# B&R Automation Studio project Ampel (part 4)

```cpp
			const TaskStatus h =
				headState.deepPreReact(control, event);
			HFSM2_IF_PLANS(region.headStatus(control) |= h);

			if (!control._consumed)
			HFSM2_IF_PLANS(region.subStatus(control) |=)
			subStates.widePreReact(control, event, active);

			return h;
		} else
	return TaskStatus{};
}

	template <typename TEvent>
	static
	HFSM2_CONSTEXPR(14)
	TaskStatus
	execute(Region& region,
			EventControl& control,
			const TEvent& event) noexcept
	{
		if (!control._consumed) {
HeadState& headState = static_cast<HeadState&>(region);
SubStates& subStates = static_cast<SubStates&>(region);

const TaskStatus h =
	headState.deepPreReact(control, event);
			HFSM2_IF_PLANS(region.headStatus(control) |= h);

			if (!control._consumed)
				HFSM2_IF_PLANS(region.subStatus(control) |=)
					subStates.widePreReact(control, event);

return h;
		} else
			return TaskStatus{};
	}

};

template <typename TRegion>
struct PreReactWrapperT<TRegion, BottomUp> {
	using Region		= TRegion;
	using HeadState		= typename Region::HeadState;
	using SubStates		= typename Region::SubStates;
	using EventControl	= typename Region::EventControl;

	template <typename TEvent>
	static
	HFSM2_CONSTEXPR(14)
	TaskStatus
	execute(Region& region,
	EventControl& control,
	const TEvent& event,
	const Prong active) noexcept
	{
	if (!control._consumed) {
	HeadState& headState = static_cast<HeadState&>(region);
	SubStates& subStates = static_cast<SubStates&>(region);

	const TaskStatus h =
		subStates.widePreReact(control, event, active);
	HFSM2_IF_PLANS(region. subStatus(control) |= h);

	if (!control._consumed)
	HFSM2_IF_PLANS(region.headStatus(control) |=)
	headState.deepPreReact(control, event);

	return h;
} else
			return TaskStatus{};
	}

	template <typename TEvent>
	static
	HFSM2_CONSTEXPR(14)
	TaskStatus
	execute(Region& region,
			EventControl& control,
			const TEvent& event) noexcept
	{
		if (!control._consumed) {
HeadState& headState = static_cast<HeadState&>(region);
SubStates& subStates = static_cast<SubStates&>(region);

const TaskStatus h =
	subStates.widePreReact(control, event);
			HFSM2_IF_PLANS(region. subStatus(control) |= h);

			if (!control._consumed)
				HFSM2_IF_PLANS(region.headStatus(control) |=)
					headState.deepPreReact(control, event);

return h;
		} else
			return TaskStatus{};
	}

};

template <typename, typename>
struct ReactWrapperT;

template <typename TRegion>
struct ReactWrapperT<TRegion, TopDown> {
	using Region		= TRegion;
	using HeadState		= typename Region::HeadState;
	using SubStates		= typename Region::SubStates;
	using EventControl	= typename Region::EventControl;

	template <typename TEvent>
	static
	HFSM2_CONSTEXPR(14)
	TaskStatus
	execute(Region& region,
	EventControl& control,
	const TEvent& event,
	const Prong active) noexcept
	{
	if (!control._consumed) {
	HeadState& headState = static_cast<HeadState&>(region);
	SubStates& subStates = static_cast<SubStates&>(region);

	const TaskStatus h =
		headState.deepReact(control, event);
	HFSM2_IF_PLANS(region.headStatus(control) |= h);

	if (!control._consumed)
	HFSM2_IF_PLANS(region. subStatus(control) |=)
	subStates.wideReact(control, event, active);

	return h;
} else
			return TaskStatus{};
	}

	template <typename TEvent>
	static
	HFSM2_CONSTEXPR(14)
	TaskStatus
	execute(Region& region,
			EventControl& control,
			const TEvent& event) noexcept
	{
		if (!control._consumed) {
HeadState& headState = static_cast<HeadState&>(region);
SubStates& subStates = static_cast<SubStates&>(region);

const TaskStatus h =
	headState.deepReact(control, event);
			HFSM2_IF_PLANS(region.headStatus(control) |= h);

			if (!control._consumed)
				HFSM2_IF_PLANS(region. subStatus(control) |=)
					subStates.wideReact(control, event);

return h;
		} else
			return TaskStatus{};
	}

};

template <typename TRegion>
struct ReactWrapperT<TRegion, BottomUp> {
	using Region		= TRegion;
	using HeadState		= typename Region::HeadState;
	using SubStates		= typename Region::SubStates;
	using EventControl	= typename Region::EventControl;

	template <typename TEvent>
	static
	HFSM2_CONSTEXPR(14)
	TaskStatus
	execute(Region& region,
	EventControl& control,
	const TEvent& event,
	const Prong active) noexcept
	{
	if (!control._consumed) {
	HeadState& headState = static_cast<HeadState&>(region);
	SubStates& subStates = static_cast<SubStates&>(region);

	const TaskStatus h =
		subStates.wideReact(control, event, active);
	HFSM2_IF_PLANS(region. subStatus(control) |= h);

	if (!control._consumed)
	HFSM2_IF_PLANS(region.headStatus(control) |=)
	headState.deepReact(control, event);

	return h;
} else
			return TaskStatus{};
	}

	template <typename TEvent>
	static
	HFSM2_CONSTEXPR(14)
	TaskStatus
	execute(Region& region,
			EventControl& control,
			const TEvent& event) noexcept
	{
		if (!control._consumed) {
HeadState& headState = static_cast<HeadState&>(region);
SubStates& subStates = static_cast<SubStates&>(region);

const TaskStatus h =
	subStates.wideReact(control, event);
			HFSM2_IF_PLANS(region. subStatus(control) |= h);

			if (!control._consumed)
				HFSM2_IF_PLANS(region.headStatus(control) |=)
					headState.deepReact(control, event);

return h;
		} else
			return TaskStatus{};
	}

};

template <typename, typename>
struct PostReactWrapperT;

template <typename TRegion>
struct PostReactWrapperT<TRegion, TopDown> {
	using Region		= TRegion;
	using HeadState		= typename Region::HeadState;
	using SubStates		= typename Region::SubStates;
	using EventControl	= typename Region::EventControl;

	template <typename TEvent>
	static
	HFSM2_CONSTEXPR(14)
	TaskStatus
	execute(Region& region,
	EventControl& control,
	const TEvent& event,
	const Prong active) noexcept
	{
	if (!control._consumed) {
	HeadState& headState = static_cast<HeadState&>(region);
	SubStates& subStates = static_cast<SubStates&>(region);

	HFSM2_IF_PLANS(region. subStatus(control) |=)
	subStates.widePostReact(control, event, active);

	if (control._consumed == false) {
	const TaskStatus h =
		headState.deepPostReact(control, event);
	HFSM2_IF_PLANS(region.headStatus(control) |= h);

	return h;
}
		}

		return TaskStatus{};
	}

	template <typename TEvent>
	static
	HFSM2_CONSTEXPR(14)
	TaskStatus
	execute(Region& region,
			EventControl& control,
			const TEvent& event) noexcept
	{
		if (!control._consumed) {
HeadState& headState = static_cast<HeadState&>(region);
SubStates& subStates = static_cast<SubStates&>(region);

			HFSM2_IF_PLANS(region. subStatus(control) |=)
				subStates.widePostReact(control, event);

			if (control._consumed == false) {
const TaskStatus h =
	headState.deepPostReact(control, event);
				HFSM2_IF_PLANS(region.headStatus(control) |= h);

return h;
			}
		}

		return TaskStatus{};
	}

};

template <typename TRegion>
struct PostReactWrapperT<TRegion, BottomUp> {
	using Region		= TRegion;
	using HeadState		= typename Region::HeadState;
	using SubStates		= typename Region::SubStates;
	using EventControl	= typename Region::EventControl;

	template <typename TEvent>
	static
	HFSM2_CONSTEXPR(14)
	TaskStatus
	execute(Region& region,
	EventControl& control,
	const TEvent& event,
	const Prong active) noexcept
	{
	if (!control._consumed) {
	HeadState& headState = static_cast<HeadState&>(region);
	SubStates& subStates = static_cast<SubStates&>(region);

	HFSM2_IF_PLANS(region.headStatus(control) |=)
	headState.deepPostReact(control, event);

	if (control._consumed == false) {
	const TaskStatus h =
		subStates.widePostReact(control, event, active);
	HFSM2_IF_PLANS(region. subStatus(control) |= h);

	return h;
}
		}

		return TaskStatus{};
	}

	template <typename TEvent>
	static
	HFSM2_CONSTEXPR(14)
	TaskStatus
	execute(Region& region,
			EventControl& control,
			const TEvent& event) noexcept
	{
		if (!control._consumed) {
HeadState& headState = static_cast<HeadState&>(region);
SubStates& subStates = static_cast<SubStates&>(region);

			HFSM2_IF_PLANS(region.headStatus(control) |=)
				headState.deepPostReact(control, event);

			if (control._consumed == false) {
const TaskStatus h =
	subStates.widePostReact(control, event);
				HFSM2_IF_PLANS(region. subStatus(control) |= h);

return h;
			}
		}

		return TaskStatus{};
	}

};

template <typename, typename>
struct QueryWrapperT;

template <typename TRegion>
struct QueryWrapperT<TRegion, TopDown> {
	using Region		= TRegion;
	using HeadState		= typename Region::HeadState;
	using SubStates		= typename Region::SubStates;
	using ConstControl	= typename Region::ConstControl;

	template <typename TEvent>
	static
	HFSM2_CONSTEXPR(14)
	void
	execute(const Region& region,
	ConstControl& control,
	TEvent& event,
	const Prong active) noexcept
	{
	const HeadState& headState = static_cast<const HeadState&>(region);
	const SubStates& subStates = static_cast<const SubStates&>(region);

	if (!control._consumed)
	headState.deepQuery(control, event);

	if (!control._consumed)
	subStates.wideQuery(control, event, active);
}

	template <typename TEvent>
	static
	HFSM2_CONSTEXPR(14)
	void
	execute(const Region& region,
			ConstControl& control,
			TEvent& event) noexcept
	{
const HeadState& headState = static_cast<const HeadState&>(region);
const SubStates& subStates = static_cast<const SubStates&>(region);

		if (!control._consumed)
			headState.deepQuery(control, event);

		if (!control._consumed)
			subStates.wideQuery(control, event);
	}

};

template <typename TRegion>
struct QueryWrapperT<TRegion, BottomUp> {
	using Region		= TRegion;
	using HeadState		= typename Region::HeadState;
	using SubStates		= typename Region::SubStates;
	using ConstControl	= typename Region::ConstControl;

	template <typename TEvent>
	static
	HFSM2_CONSTEXPR(14)
	void
	execute(const Region& region,
	ConstControl& control,
	TEvent& event,
	const Prong active) noexcept
	{
	const HeadState& headState = static_cast<const HeadState&>(region);
	const SubStates& subStates = static_cast<const SubStates&>(region);

	if (!control._consumed)
	subStates.wideQuery(control, event, active);

	if (!control._consumed)
	headState.deepQuery(control, event);
}

	template <typename TEvent>
	static
	HFSM2_CONSTEXPR(14)
	void
	execute(const Region& region,
			ConstControl& control,
			TEvent& event) noexcept
	{
const HeadState& headState = static_cast<const HeadState&>(region);
const SubStates& subStates = static_cast<const SubStates&>(region);

		if (!control._consumed)
			subStates.wideQuery(control, event);

		if (!control._consumed)
			headState.deepQuery(control, event);
	}

};

}
}

namespace hfsm2 {
	namespace detail {

		template <
		typename TIndices
		, typename TArgs
		, Strategy TStrategy
		, Prong NProng
		, typename... TStates
		>
		struct HFSM2_EMPTY_BASES CS_<
			TIndices
			, TArgs
			, TStrategy
			, NProng
			, TL_<TStates...>
		>
		:					 LHalfCS<
		TIndices
		, TArgs
		, TStrategy
		, NProng
		, TL_<TStates...>
		>
		,					 RHalfCS<
		TIndices
		, TArgs
		, TStrategy
		, NProng
		, TL_<TStates...>
		>
		{
		static_assert(sizeof...(TStates) >= 2, "");

		using Indices		= TIndices;
		static constexpr StateID  INITIAL_ID  = Indices::STATE_ID;
		static constexpr Short	  COMPO_INDEX = Indices::COMPO_INDEX;
		static constexpr Short	  ORTHO_INDEX = Indices::ORTHO_INDEX;
		static constexpr Short	  ORTHO_UNIT  = Indices::ORTHO_UNIT;

		static constexpr Strategy STRATEGY	  = TStrategy;

		static constexpr RegionID REGION_ID	  = COMPO_INDEX + ORTHO_INDEX;
		static constexpr Prong	  PRONG_INDEX = NProng;

		using Args			= TArgs;
		using SubStateList	= TL_<TStates...>;

#if HFSM2_UTILITY_THEORY_AVAILABLE()
		using Rank			= typename Args::Rank;
		using Utility		= typename Args::Utility;
		using UP			= typename Args::UP;
#endif

		using StateList		= typename Args::StateList;
		using RegionList	= typename Args::RegionList;

		using Registry		= RegistryT<Args>;
		using StateParents	= typename Registry::StateParents;

		using ConstControl	= ConstControlT<Args>;
		using Control		= ControlT	   <Args>;
		using PlanControl	= PlanControlT <Args>;
		using FullControl	= FullControlT <Args>;
		using GuardControl	= GuardControlT<Args>;
		using EventControl	= EventControlT<Args>;

		using LStateList	= LHalfTypes<TStates...>;
		using LHalfInfo		= CSI_<LStateList>;

		static constexpr Prong	  L_PRONG	  = PRONG_INDEX;
		static constexpr Prong	  R_PRONG	  = PRONG_INDEX + LStateList::SIZE;

		using LHalf			= LHalfCS<
			Indices
			, Args
			, STRATEGY
			, PRONG_INDEX
			, SubStateList
			>;

		using RHalf			= RHalfCS<
			Indices
			, Args
			, STRATEGY
			, PRONG_INDEX
			, SubStateList
			>;

		HFSM2_CONSTEXPR(14)	void		wideRegister			   (Registry& registry, const Parent parent)								noexcept;

		HFSM2_CONSTEXPR(14)	bool		wideForwardEntryGuard	   (GuardControl& control,						  const Prong prong)		noexcept;
		HFSM2_CONSTEXPR(14)	bool		wideEntryGuard			   (GuardControl& control,						  const Prong prong)		noexcept;

		HFSM2_CONSTEXPR(14)	void		wideEnter				   ( PlanControl& control,						  const Prong prong)		noexcept;
		HFSM2_CONSTEXPR(14)	void		wideReenter				   ( PlanControl& control,						  const Prong prong)		noexcept;

		HFSM2_CONSTEXPR(14)	TaskStatus	widePreUpdate			   ( FullControl& control,						  const Prong prong)		noexcept;
		HFSM2_CONSTEXPR(14)	TaskStatus	wideUpdate				   ( FullControl& control,						  const Prong prong)		noexcept;
		HFSM2_CONSTEXPR(14)	TaskStatus	widePostUpdate			   ( FullControl& control,						  const Prong prong)		noexcept;

		template <typename TEvent>
		HFSM2_CONSTEXPR(14)	TaskStatus	widePreReact			   (EventControl& control, const TEvent& event,	  const Prong prong)		noexcept;

		template <typename TEvent>
		HFSM2_CONSTEXPR(14)	TaskStatus	wideReact				   (EventControl& control, const TEvent& event,	  const Prong prong)		noexcept;

		template <typename TEvent>
		HFSM2_CONSTEXPR(14)	TaskStatus	widePostReact			   (EventControl& control, const TEvent& event,	  const Prong prong)		noexcept;

		template <typename TEvent>
		HFSM2_CONSTEXPR(14)	void		wideQuery				   (ConstControl& control,		 TEvent& event,	  const Prong prong)  const noexcept;

#if HFSM2_PLANS_AVAILABLE()
		HFSM2_CONSTEXPR(14)	TaskStatus	wideUpdatePlans			   ( FullControl& control,						  const Prong prong)		noexcept;
#endif

		HFSM2_CONSTEXPR(14)	bool		wideForwardExitGuard	   (GuardControl& control,						  const Prong prong)		noexcept;
		HFSM2_CONSTEXPR(14)	bool		wideExitGuard			   (GuardControl& control,						  const Prong prong)		noexcept;

		HFSM2_CONSTEXPR(14)	void		wideExit				   ( PlanControl& control,						  const Prong prong)		noexcept;

		HFSM2_CONSTEXPR(14)	void		wideForwardActive		   (	 Control& control, const Request request, const Prong prong)		noexcept;
		HFSM2_CONSTEXPR(14)	void		wideForwardRequest		   (	 Control& control, const Request request, const Prong prong)		noexcept;

		HFSM2_CONSTEXPR(14)	void		wideRequestChangeComposite (	 Control& control, const Request request				   )		noexcept;
		HFSM2_CONSTEXPR(14)	void		wideRequestChangeResumable (	 Control& control, const Request request, const Prong prong)		noexcept;
		HFSM2_CONSTEXPR(14)	void		wideRequestChangeSelectable(	 Control& control, const Request request, const Prong prong)		noexcept;

		HFSM2_CONSTEXPR(14)	void		wideRequestRestart		   (	 Control& control, const Request request				   )		noexcept;
		HFSM2_CONSTEXPR(14)	void		wideRequestResume		   (	 Control& control, const Request request, const Prong prong)		noexcept;
		HFSM2_CONSTEXPR(14)	void		wideRequestSelect		   (	 Control& control, const Request request, const Prong prong)		noexcept;

#if HFSM2_UTILITY_THEORY_AVAILABLE()
		HFSM2_CONSTEXPR(14)	UP			wideReportChangeComposite  (	 Control& control																  )		noexcept;
		HFSM2_CONSTEXPR(14)	UP			wideReportChangeResumable  (	 Control& control,						  const Prong prong						  )		noexcept;
		HFSM2_CONSTEXPR(14)	UP			wideReportChangeSelectable (	 Control& control,						  const Prong prong						  )		noexcept;
		HFSM2_CONSTEXPR(14)	UP			wideReportChangeUtilitarian(	 Control& control																  )		noexcept;
		HFSM2_CONSTEXPR(14)	Utility		wideReportChangeRandom	   (	 Control& control, Utility* const options, const Rank* const ranks, const Rank top)		noexcept;

		HFSM2_CONSTEXPR(14)	UP			wideReportUtilize		   (	 Control& control																  )		noexcept;
		HFSM2_CONSTEXPR(14)	Rank		wideReportRank			   (	 Control& control,								 Rank* const ranks				  )		noexcept;
		HFSM2_CONSTEXPR(14)	Utility		wideReportRandomize		   (	 Control& control, Utility* const options, const Rank* const ranks, const Rank top)		noexcept;
#endif

		HFSM2_CONSTEXPR(14)	void		wideChangeToRequested	   ( PlanControl& control,						  const Prong prong)		noexcept;

#if HFSM2_SERIALIZATION_AVAILABLE()
		using WriteStream	= typename Args::WriteStream;
		using ReadStream	= typename Args::ReadStream;

		HFSM2_CONSTEXPR(14)	void		wideSaveActive			   (const Registry& registry, WriteStream& stream, const Prong prong)  const noexcept;
		HFSM2_CONSTEXPR(14)	void		wideSaveResumable		   (const Registry& registry, WriteStream& stream					)  const noexcept;

		HFSM2_CONSTEXPR(14)	void		wideLoadRequested		   (      Registry& registry,  ReadStream& stream, const Prong prong)  const noexcept;
		HFSM2_CONSTEXPR(14)	void		wideLoadResumable		   (      Registry& registry,  ReadStream& stream					)  const noexcept;
#endif

#if HFSM2_STRUCTURE_REPORT_AVAILABLE()
		using StructureStateInfos = typename Args::StructureStateInfos;

		static constexpr Long NAME_COUNT = LHalf::NAME_COUNT + RHalf::NAME_COUNT;

		HFSM2_CONSTEXPR(14)	void wideGetNames(const Long parent,
		const RegionType region,
		const Short depth,
		StructureStateInfos& stateInfos)	  const noexcept;
#endif

	};

}
}

namespace hfsm2 {
	namespace detail {

		template <typename TN_, typename TA_, Strategy SG_, Prong NP_, typename... TS_>
		HFSM2_CONSTEXPR(14)
		void
			CS_<TN_, TA_, SG_, NP_, TL_<TS_...>>::wideRegister(Registry& registry,
		const Parent parent) noexcept
		{
		LHalf::wideRegister(registry, Parent{parent.forkId, L_PRONG});
		RHalf::wideRegister(registry, Parent{parent.forkId, R_PRONG});
	}

	template <typename TN_, typename TA_, Strategy SG_, Prong NP_, typename... TS_>
	HFSM2_CONSTEXPR(14)
	bool
		CS_<TN_, TA_, SG_, NP_, TL_<TS_...>>::wideForwardEntryGuard(GuardControl& control,
	const Prong prong) noexcept
	{
	HFSM2_ASSERT(prong != INVALID_SHORT);

	if (prong < R_PRONG)
	return LHalf::wideForwardEntryGuard(control, prong);
	else
	return RHalf::wideForwardEntryGuard(control, prong);
}

template <typename TN_, typename TA_, Strategy SG_, Prong NP_, typename... TS_>
HFSM2_CONSTEXPR(14)
bool
	CS_<TN_, TA_, SG_, NP_, TL_<TS_...>>::wideEntryGuard(GuardControl& control,
													 const Prong prong) noexcept
{
	HFSM2_ASSERT(prong != INVALID_PRONG);

	if (prong < R_PRONG)
		return LHalf::wideEntryGuard(control, prong);
	else
		return RHalf::wideEntryGuard(control, prong);
}

template <typename TN_, typename TA_, Strategy SG_, Prong NP_, typename... TS_>
HFSM2_CONSTEXPR(14)
void
	CS_<TN_, TA_, SG_, NP_, TL_<TS_...>>::wideEnter(PlanControl& control,
												const Prong prong) noexcept
{
	HFSM2_ASSERT(prong != INVALID_PRONG);

	if (prong < R_PRONG)
		LHalf::wideEnter(control, prong);
	else
		RHalf::wideEnter(control, prong);
}

template <typename TN_, typename TA_, Strategy SG_, Prong NP_, typename... TS_>
HFSM2_CONSTEXPR(14)
void
	CS_<TN_, TA_, SG_, NP_, TL_<TS_...>>::wideReenter(PlanControl& control,
												  const Prong prong) noexcept
{
	HFSM2_ASSERT(prong != INVALID_PRONG);

	if (prong < R_PRONG)
		LHalf::wideReenter(control, prong);
	else
		RHalf::wideReenter(control, prong);
}

template <typename TN_, typename TA_, Strategy SG_, Prong NP_, typename... TS_>
HFSM2_CONSTEXPR(14)
TaskStatus
	CS_<TN_, TA_, SG_, NP_, TL_<TS_...>>::widePreUpdate(FullControl& control,
													const Prong prong) noexcept
{
	HFSM2_ASSERT(prong != INVALID_PRONG);

	return prong < R_PRONG ?
		LHalf::widePreUpdate(control, prong) :
		RHalf::widePreUpdate(control, prong);
}

template <typename TN_, typename TA_, Strategy SG_, Prong NP_, typename... TS_>
HFSM2_CONSTEXPR(14)
TaskStatus
	CS_<TN_, TA_, SG_, NP_, TL_<TS_...>>::wideUpdate(FullControl& control,
												 const Prong prong) noexcept
{
	HFSM2_ASSERT(prong != INVALID_PRONG);

	return prong < R_PRONG ?
		LHalf::wideUpdate(control, prong) :
		RHalf::wideUpdate(control, prong);
}

template <typename TN_, typename TA_, Strategy SG_, Prong NP_, typename... TS_>
HFSM2_CONSTEXPR(14)
TaskStatus
	CS_<TN_, TA_, SG_, NP_, TL_<TS_...>>::widePostUpdate(FullControl& control,
													 const Prong prong) noexcept
{
	HFSM2_ASSERT(prong != INVALID_PRONG);

	return prong < R_PRONG ?
		LHalf::widePostUpdate(control, prong) :
		RHalf::widePostUpdate(control, prong);
}

template <typename TN_, typename TA_, Strategy SG_, Prong NP_, typename... TS_>
template <typename TEvent>
HFSM2_CONSTEXPR(14)
TaskStatus
	CS_<TN_, TA_, SG_, NP_, TL_<TS_...>>::widePreReact(EventControl& control,
												   const TEvent& event,
												   const Prong prong) noexcept
{
	HFSM2_ASSERT(prong != INVALID_PRONG);

	return prong < R_PRONG ?
		LHalf::widePreReact(control, event, prong) :
		RHalf::widePreReact(control, event, prong);
}

template <typename TN_, typename TA_, Strategy SG_, Prong NP_, typename... TS_>
template <typename TEvent>
HFSM2_CONSTEXPR(14)
TaskStatus
	CS_<TN_, TA_, SG_, NP_, TL_<TS_...>>::wideReact(EventControl& control,
												const TEvent& event,
												const Prong prong) noexcept
{
	HFSM2_ASSERT(prong != INVALID_PRONG);

	return prong < R_PRONG ?
		LHalf::wideReact(control, event, prong) :
		RHalf::wideReact(control, event, prong);
}

template <typename TN_, typename TA_, Strategy SG_, Prong NP_, typename... TS_>
template <typename TEvent>
HFSM2_CONSTEXPR(14)
TaskStatus
	CS_<TN_, TA_, SG_, NP_, TL_<TS_...>>::widePostReact(EventControl& control,
													const TEvent& event,
													const Prong prong) noexcept
{
	HFSM2_ASSERT(prong != INVALID_PRONG);

	return prong < R_PRONG ?
		LHalf::widePostReact(control, event, prong) :
		RHalf::widePostReact(control, event, prong);
}

template <typename TN_, typename TA_, Strategy SG_, Prong NP_, typename... TS_>
template <typename TEvent>
HFSM2_CONSTEXPR(14)
void
	CS_<TN_, TA_, SG_, NP_, TL_<TS_...>>::wideQuery(ConstControl& control,
												TEvent& event,
												const Prong prong) const noexcept
{
	HFSM2_ASSERT(prong != INVALID_PRONG);

	return prong < R_PRONG ?
		LHalf::wideQuery(control, event, prong) :
		RHalf::wideQuery(control, event, prong);
}

#if HFSM2_PLANS_AVAILABLE()

template <typename TN_, typename TA_, Strategy SG_, Prong NP_, typename... TS_>
HFSM2_CONSTEXPR(14)
TaskStatus
	CS_<TN_, TA_, SG_, NP_, TL_<TS_...>>::wideUpdatePlans(FullControl& control,
													  const Prong prong) noexcept
{
	HFSM2_ASSERT(prong != INVALID_PRONG);

	return prong < R_PRONG ?
		LHalf::wideUpdatePlans(control, prong) :
		RHalf::wideUpdatePlans(control, prong);
}

#endif

template <typename TN_, typename TA_, Strategy SG_, Prong NP_, typename... TS_>
HFSM2_CONSTEXPR(14)
bool
	CS_<TN_, TA_, SG_, NP_, TL_<TS_...>>::wideForwardExitGuard(GuardControl& control,
														   const Prong prong) noexcept
{
	HFSM2_ASSERT(prong != INVALID_PRONG);

	if (prong < R_PRONG)
		return LHalf::wideForwardExitGuard(control, prong);
	else
		return RHalf::wideForwardExitGuard(control, prong);
}

template <typename TN_, typename TA_, Strategy SG_, Prong NP_, typename... TS_>
HFSM2_CONSTEXPR(14)
bool
	CS_<TN_, TA_, SG_, NP_, TL_<TS_...>>::wideExitGuard(GuardControl& control,
													const Prong prong) noexcept
{
	HFSM2_ASSERT(prong != INVALID_PRONG);

	if (prong < R_PRONG)
		return LHalf::wideExitGuard(control, prong);
	else
		return RHalf::wideExitGuard(control, prong);
}

template <typename TN_, typename TA_, Strategy SG_, Prong NP_, typename... TS_>
HFSM2_CONSTEXPR(14)
void
	CS_<TN_, TA_, SG_, NP_, TL_<TS_...>>::wideExit(PlanControl& control,
											   const Prong prong) noexcept
{
	HFSM2_ASSERT(prong != INVALID_PRONG);

	if (prong < R_PRONG)
		LHalf::wideExit(control, prong);
	else
		RHalf::wideExit(control, prong);
}

template <typename TN_, typename TA_, Strategy SG_, Prong NP_, typename... TS_>
HFSM2_CONSTEXPR(14)
void
	CS_<TN_, TA_, SG_, NP_, TL_<TS_...>>::wideForwardActive(Control& control,
														const Request request,
														const Prong prong) noexcept
{
	HFSM2_ASSERT(prong != INVALID_PRONG);

	if (prong < R_PRONG)
		LHalf::wideForwardActive(control, request, prong);
	else
		RHalf::wideForwardActive(control, request, prong);
}

template <typename TN_, typename TA_, Strategy SG_, Prong NP_, typename... TS_>
HFSM2_CONSTEXPR(14)
void
	CS_<TN_, TA_, SG_, NP_, TL_<TS_...>>::wideForwardRequest(Control& control,
														 const Request request,
														 const Prong prong) noexcept
{
	HFSM2_ASSERT(prong != INVALID_PRONG);

	if (prong < R_PRONG)
		LHalf::wideForwardRequest(control, request, prong);
	else
		RHalf::wideForwardRequest(control, request, prong);
}

template <typename TN_, typename TA_, Strategy SG_, Prong NP_, typename... TS_>
HFSM2_CONSTEXPR(14)
void
	CS_<TN_, TA_, SG_, NP_, TL_<TS_...>>::wideRequestChangeComposite(Control& control,
																 const Request request) noexcept
{
	LHalf::wideRequestChangeComposite(control, request);
}

template <typename TN_, typename TA_, Strategy SG_, Prong NP_, typename... TS_>
HFSM2_CONSTEXPR(14)
void
	CS_<TN_, TA_, SG_, NP_, TL_<TS_...>>::wideRequestChangeResumable(Control& control,
																 const Request request,
																 const Prong prong) noexcept
{
	HFSM2_ASSERT(prong != INVALID_PRONG);

	if (prong < R_PRONG)
		LHalf::wideRequestChangeResumable(control, request, prong);
	else
		RHalf::wideRequestChangeResumable(control, request, prong);
}

template <typename TN_, typename TA_, Strategy SG_, Prong NP_, typename... TS_>
HFSM2_CONSTEXPR(14)
void
	CS_<TN_, TA_, SG_, NP_, TL_<TS_...>>::wideRequestChangeSelectable(Control& control,
																  const Request request,
																  const Prong prong) noexcept
{
	HFSM2_ASSERT(prong != INVALID_PRONG);

	if (prong < R_PRONG)
		LHalf::wideRequestChangeSelectable(control, request, prong);
	else
		RHalf::wideRequestChangeSelectable(control, request, prong);
}

template <typename TN_, typename TA_, Strategy SG_, Prong NP_, typename... TS_>
HFSM2_CONSTEXPR(14)
void
	CS_<TN_, TA_, SG_, NP_, TL_<TS_...>>::wideRequestRestart(Control& control,
														 const Request request) noexcept
{
	LHalf::wideRequestRestart(control, request);
}

template <typename TN_, typename TA_, Strategy SG_, Prong NP_, typename... TS_>
HFSM2_CONSTEXPR(14)
void
	CS_<TN_, TA_, SG_, NP_, TL_<TS_...>>::wideRequestResume(Control& control,
														const Request request,
														const Prong prong) noexcept
{
	HFSM2_ASSERT(prong != INVALID_PRONG);

	if (prong < R_PRONG)
		LHalf::wideRequestResume(control, request, prong);
	else
		RHalf::wideRequestResume(control, request, prong);
}

template <typename TN_, typename TA_, Strategy SG_, Prong NP_, typename... TS_>
HFSM2_CONSTEXPR(14)
void
	CS_<TN_, TA_, SG_, NP_, TL_<TS_...>>::wideRequestSelect(Control& control,
														const Request request,
														const Prong prong) noexcept
{
	HFSM2_ASSERT(prong != INVALID_PRONG);

	if (prong < R_PRONG)
		LHalf::wideRequestSelect(control, request, prong);
	else
		RHalf::wideRequestSelect(control, request, prong);
}

#if HFSM2_UTILITY_THEORY_AVAILABLE()

template <typename TN_, typename TA_, Strategy SG_, Prong NP_, typename... TS_>
HFSM2_CONSTEXPR(14)
typename TA_::UP
	CS_<TN_, TA_, SG_, NP_, TL_<TS_...>>::wideReportUtilize(Control& control) noexcept {
const UP l = LHalf::wideReportUtilize(control);
const UP r = RHalf::wideReportUtilize(control);

	return l.utility >= r.utility ?
l : r;
}

template <typename TN_, typename TA_, Strategy SG_, Prong NP_, typename... TS_>
HFSM2_CONSTEXPR(14)
typename TA_::Rank
	CS_<TN_, TA_, SG_, NP_, TL_<TS_...>>::wideReportRank(Control& control,
													 Rank* const ranks) noexcept
{
	HFSM2_ASSERT(ranks);

const Rank l = LHalf::wideReportRank(control, ranks);
const Rank r = RHalf::wideReportRank(control, ranks + LStateList::SIZE);

	return l >= r ?
l : r;
}

template <typename TN_, typename TA_, Strategy SG_, Prong NP_, typename... TS_>
HFSM2_CONSTEXPR(14)
typename TA_::Utility
	CS_<TN_, TA_, SG_, NP_, TL_<TS_...>>::wideReportRandomize(Control& control,
														  Utility* const utilities,
														  const Rank* const ranks,
														  const Rank top) noexcept
{
	HFSM2_ASSERT(utilities && ranks);

const Utility l = LHalf::wideReportRandomize(control, utilities,					ranks,					  top);
const Utility r = RHalf::wideReportRandomize(control, utilities + LStateList::SIZE, ranks + LStateList::SIZE, top);

	return { l + r };
}

template <typename TN_, typename TA_, Strategy SG_, Prong NP_, typename... TS_>
HFSM2_CONSTEXPR(14)
typename TA_::UP
	CS_<TN_, TA_, SG_, NP_, TL_<TS_...>>::wideReportChangeComposite(Control& control) noexcept {
	return LHalf::wideReportChangeComposite(control);
}

template <typename TN_, typename TA_, Strategy SG_, Prong NP_, typename... TS_>
HFSM2_CONSTEXPR(14)
typename TA_::UP
	CS_<TN_, TA_, SG_, NP_, TL_<TS_...>>::wideReportChangeResumable(Control& control,
																const Prong prong) noexcept
{
	HFSM2_ASSERT(prong != INVALID_PRONG);

	if (prong < R_PRONG)
		return LHalf::wideReportChangeResumable(control, prong);
	else
		return RHalf::wideReportChangeResumable(control, prong);
}

template <typename TN_, typename TA_, Strategy SG_, Prong NP_, typename... TS_>
HFSM2_CONSTEXPR(14)
typename TA_::UP
	CS_<TN_, TA_, SG_, NP_, TL_<TS_...>>::wideReportChangeSelectable(Control& control,
																 const Prong prong) noexcept
{
	HFSM2_ASSERT(prong != INVALID_PRONG);

	if (prong < R_PRONG)
		return LHalf::wideReportChangeSelectable(control, prong);
	else
		return RHalf::wideReportChangeSelectable(control, prong);
}

template <typename TN_, typename TA_, Strategy SG_, Prong NP_, typename... TS_>
HFSM2_CONSTEXPR(14)
typename TA_::UP
	CS_<TN_, TA_, SG_, NP_, TL_<TS_...>>::wideReportChangeUtilitarian(Control& control) noexcept {
const UP l = LHalf::wideReportChangeUtilitarian(control);
const UP r = RHalf::wideReportChangeUtilitarian(control);

	return l.utility >= r.utility ?
l : r;
}

template <typename TN_, typename TA_, Strategy SG_, Prong NP_, typename... TS_>
HFSM2_CONSTEXPR(14)
typename TA_::Utility
	CS_<TN_, TA_, SG_, NP_, TL_<TS_...>>::wideReportChangeRandom(Control& control,
															 Utility* const utilities,
															 const Rank* const ranks,
															 const Rank top) noexcept
{
	HFSM2_ASSERT(utilities && ranks);

const Utility l = LHalf::wideReportChangeRandom(control, utilities,					   ranks,					 top);
const Utility r = RHalf::wideReportChangeRandom(control, utilities + LStateList::SIZE, ranks + LStateList::SIZE, top);

	return { l + r };
}

#endif

template <typename TN_, typename TA_, Strategy SG_, Prong NP_, typename... TS_>
HFSM2_CONSTEXPR(14)
void
	CS_<TN_, TA_, SG_, NP_, TL_<TS_...>>::wideChangeToRequested(PlanControl& control,
															const Prong prong) noexcept
{
	HFSM2_ASSERT(prong != INVALID_PRONG);

	if (prong < R_PRONG)
		LHalf::wideChangeToRequested(control, prong);
	else
		RHalf::wideChangeToRequested(control, prong);
}

#if HFSM2_SERIALIZATION_AVAILABLE()

template <typename TN_, typename TA_, Strategy SG_, Prong NP_, typename... TS_>
HFSM2_CONSTEXPR(14)
void
	CS_<TN_, TA_, SG_, NP_, TL_<TS_...>>::wideSaveActive(const Registry& registry,
													 WriteStream& stream,
													 const Prong prong) const noexcept
{
	HFSM2_ASSERT(prong != INVALID_PRONG);

	if (prong < R_PRONG) {
		LHalf::wideSaveActive   (registry, stream, prong);
		RHalf::wideSaveResumable(registry, stream);
	} else {
		LHalf::wideSaveResumable(registry, stream);
		RHalf::wideSaveActive   (registry, stream, prong);
	}
}

template <typename TN_, typename TA_, Strategy SG_, Prong NP_, typename... TS_>
HFSM2_CONSTEXPR(14)
void
	CS_<TN_, TA_, SG_, NP_, TL_<TS_...>>::wideSaveResumable(const Registry& registry,
														WriteStream& stream) const noexcept
{
	LHalf::wideSaveResumable(registry, stream);
	RHalf::wideSaveResumable(registry, stream);
}

template <typename TN_, typename TA_, Strategy SG_, Prong NP_, typename... TS_>
HFSM2_CONSTEXPR(14)
void
	CS_<TN_, TA_, SG_, NP_, TL_<TS_...>>::wideLoadRequested(Registry& registry,
														ReadStream& stream,
														const Prong prong) const noexcept
{
	HFSM2_ASSERT(prong != INVALID_PRONG);

	if (prong < R_PRONG) {
		LHalf::wideLoadRequested(registry, stream, prong);
		RHalf::wideLoadResumable(registry, stream);
	} else {
		LHalf::wideLoadResumable(registry, stream);
		RHalf::wideLoadRequested(registry, stream, prong);
	}
}

template <typename TN_, typename TA_, Strategy SG_, Prong NP_, typename... TS_>
HFSM2_CONSTEXPR(14)
void
	CS_<TN_, TA_, SG_, NP_, TL_<TS_...>>::wideLoadResumable(Registry& registry,
														ReadStream& stream) const noexcept
{
	LHalf::wideLoadResumable(registry, stream);
	RHalf::wideLoadResumable(registry, stream);
}

#endif

#if HFSM2_STRUCTURE_REPORT_AVAILABLE()

template <typename TN_, typename TA_, Strategy SG_, Prong NP_, typename... TS_>
HFSM2_CONSTEXPR(14)
void
	CS_<TN_, TA_, SG_, NP_, TL_<TS_...>>::wideGetNames(const Long parent,
												   const RegionType /*region*/,
												   const Short depth,
												   StructureStateInfos& stateInfos) const noexcept
{
	LHalf::wideGetNames(parent, RegionType::COMPOSITE, depth, stateInfos);
	RHalf::wideGetNames(parent, RegionType::COMPOSITE, depth, stateInfos);
}

#endif

}
}

namespace hfsm2 {
	namespace detail {

		template <
		typename TIndices
		, typename TArgs
		, Strategy TStrategy
		, Prong NProng
		, typename TState
		>
		struct HFSM2_EMPTY_BASES CS_<
			TIndices
			, TArgs
			, TStrategy
			, NProng
			, TL_<TState>
			>
			:					 MaterialT<
			TIndices
			, TArgs
			, TState
			>
			{
			using Indices		= TIndices;
			static constexpr StateID  INITIAL_ID  = Indices::STATE_ID;
			static constexpr Short	  COMPO_INDEX = Indices::COMPO_INDEX;
			static constexpr Short	  ORTHO_INDEX = Indices::ORTHO_INDEX;
			static constexpr Short	  ORTHO_UNIT  = Indices::ORTHO_UNIT;

			static constexpr Strategy STRATEGY	  = TStrategy;

			static constexpr RegionID REGION_ID	  = COMPO_INDEX + ORTHO_INDEX;
			static constexpr Prong	  PRONG_INDEX = NProng;

			using Args			= TArgs;

#if HFSM2_UTILITY_THEORY_AVAILABLE()
			using Rank			= typename Args::Rank;
			using Utility		= typename Args::Utility;
			using UP			= typename Args::UP;
#endif

			using StateList		= typename Args::StateList;
			using RegionList	= typename Args::RegionList;

			using Registry		= RegistryT<Args>;
			using StateParents	= typename Registry::StateParents;

			using ConstControl	= ConstControlT<Args>;
			using Control		= ControlT	   <Args>;
			using PlanControl	= PlanControlT <Args>;
			using FullControl	= FullControlT <Args>;
			using GuardControl	= GuardControlT<Args>;
			using EventControl	= EventControlT<Args>;

			using Single		= MaterialT<
				Indices
				, Args
				, TState
				>;

			HFSM2_CONSTEXPR(14)	void		wideRegister			   (Registry& registry, const Parent parent)								noexcept;

			HFSM2_CONSTEXPR(14)	bool		wideForwardEntryGuard	   (GuardControl& control,						  const Prong prong)		noexcept;
			HFSM2_CONSTEXPR(14)	bool		wideEntryGuard			   (GuardControl& control,						  const Prong prong)		noexcept;

			HFSM2_CONSTEXPR(14)	void		wideEnter				   ( PlanControl& control,						  const Prong prong)		noexcept;
			HFSM2_CONSTEXPR(14)	void		wideReenter				   ( PlanControl& control,						  const Prong prong)		noexcept;

			HFSM2_CONSTEXPR(14)	TaskStatus	widePreUpdate			   ( FullControl& control,						  const Prong prong)		noexcept;
			HFSM2_CONSTEXPR(14)	TaskStatus	wideUpdate				   ( FullControl& control,						  const Prong prong)		noexcept;
			HFSM2_CONSTEXPR(14)	TaskStatus	widePostUpdate			   ( FullControl& control,						  const Prong prong)		noexcept;

			template <typename TEvent>
			HFSM2_CONSTEXPR(14)	TaskStatus	widePreReact			   (EventControl& control, const TEvent& event,	  const Prong prong)		noexcept;

			template <typename TEvent>
			HFSM2_CONSTEXPR(14)	TaskStatus	wideReact				   (EventControl& control, const TEvent& event,	  const Prong prong)		noexcept;

			template <typename TEvent>
			HFSM2_CONSTEXPR(14)	TaskStatus	widePostReact			   (EventControl& control, const TEvent& event,	  const Prong prong)		noexcept;

			template <typename TEvent>
			HFSM2_CONSTEXPR(14)	void		wideQuery				   (ConstControl& control,		 TEvent& event,	  const Prong prong)  const noexcept;

#if HFSM2_PLANS_AVAILABLE()
			HFSM2_CONSTEXPR(14)	TaskStatus	wideUpdatePlans			   ( FullControl& control,						  const Prong prong)		noexcept;
#endif

			HFSM2_CONSTEXPR(14)	bool		wideForwardExitGuard	   (GuardControl& control,						  const Prong prong)		noexcept;
			HFSM2_CONSTEXPR(14)	bool		wideExitGuard			   (GuardControl& control,						  const Prong prong)		noexcept;

			HFSM2_CONSTEXPR(14)	void		wideExit				   ( PlanControl& control,						  const Prong prong)		noexcept;

			HFSM2_CONSTEXPR(14)	void		wideForwardActive		   (	 Control& control, const Request request, const Prong prong)		noexcept;
			HFSM2_CONSTEXPR(14)	void		wideForwardRequest		   (	 Control& control, const Request request, const Prong prong)		noexcept;

			HFSM2_CONSTEXPR(14)	void		wideRequestChangeComposite (	 Control& control, const Request request				   )		noexcept;
			HFSM2_CONSTEXPR(14)	void		wideRequestChangeResumable (	 Control& control, const Request request, const Prong prong)		noexcept;
			HFSM2_CONSTEXPR(14)	void		wideRequestChangeSelectable(	 Control& control, const Request request, const Prong prong)		noexcept;

			HFSM2_CONSTEXPR(14)	void		wideRequestRestart		   (	 Control& control, const Request request				   )		noexcept;
			HFSM2_CONSTEXPR(14)	void		wideRequestResume		   (	 Control& control, const Request request, const Prong prong)		noexcept;
			HFSM2_CONSTEXPR(14)	void		wideRequestSelect		   (	 Control& control, const Request request, const Prong prong)		noexcept;

#if HFSM2_UTILITY_THEORY_AVAILABLE()
			HFSM2_CONSTEXPR(14)	UP			wideReportChangeComposite  (	 Control& control																  )		noexcept;
			HFSM2_CONSTEXPR(14)	UP			wideReportChangeResumable  (	 Control& control						, const Prong prong						  )		noexcept;
			HFSM2_CONSTEXPR(14)	UP			wideReportChangeSelectable (	 Control& control						, const Prong prong						  )		noexcept;
			HFSM2_CONSTEXPR(14)	UP			wideReportChangeUtilitarian(	 Control& control																  )		noexcept;
			HFSM2_CONSTEXPR(14)	Utility		wideReportChangeRandom	   (	 Control& control, Utility* const options, const Rank* const ranks, const Rank top)		noexcept;

			HFSM2_CONSTEXPR(14)	UP			wideReportUtilize		   (	 Control& control																  )		noexcept;
			HFSM2_CONSTEXPR(14)	Rank		wideReportRank			   (	 Control& control,								 Rank* const ranks				  )		noexcept;
			HFSM2_CONSTEXPR(14)	Utility		wideReportRandomize		   (	 Control& control, Utility* const options, const Rank* const ranks, const Rank top)		noexcept;
#endif

			HFSM2_CONSTEXPR(14)	void		wideChangeToRequested	   ( PlanControl& control,						  const Prong prong)		noexcept;

#if HFSM2_SERIALIZATION_AVAILABLE()
			using WriteStream	= typename Args::WriteStream;
			using ReadStream	= typename Args::ReadStream;

			HFSM2_CONSTEXPR(14)	void		wideSaveActive			   (const Registry& registry, WriteStream& stream, const Prong prong)  const noexcept;
			HFSM2_CONSTEXPR(14)	void		wideSaveResumable		   (const Registry& registry, WriteStream& stream					)  const noexcept;

			HFSM2_CONSTEXPR(14)	void		wideLoadRequested		   (      Registry& registry,  ReadStream& stream, const Prong prong)  const noexcept;
			HFSM2_CONSTEXPR(14)	void		wideLoadResumable		   (      Registry& registry,  ReadStream& stream					)  const noexcept;
#endif

#if HFSM2_STRUCTURE_REPORT_AVAILABLE()
			using StructureStateInfos = typename Args::StructureStateInfos;

			static constexpr Long NAME_COUNT = Single::NAME_COUNT;

			HFSM2_CONSTEXPR(14)	void wideGetNames(const Long parent,
			const RegionType region,
			const Short depth,
			StructureStateInfos& stateInfos)	  const noexcept;
#endif

		};

	}
}

namespace hfsm2 {
	namespace detail {

		template <typename TN_, typename TA_, Strategy SG_, Prong NP_, typename T_>
		HFSM2_CONSTEXPR(14)
		void
		CS_<TN_, TA_, SG_, NP_, TL_<T_>>::wideRegister(Registry& registry,
		const Parent parent) noexcept
		{
		Single::deepRegister(registry, Parent{parent.forkId, PRONG_INDEX});
	}

	template <typename TN_, typename TA_, Strategy SG_, Prong NP_, typename T_>
	HFSM2_CONSTEXPR(14)
	bool
	CS_<TN_, TA_, SG_, NP_, TL_<T_>>::wideForwardEntryGuard(GuardControl& control,
	const Prong HFSM2_IF_ASSERT(prong)) noexcept
	{
	HFSM2_ASSERT(prong == PRONG_INDEX);

	return Single::deepForwardEntryGuard(control);
}

template <typename TN_, typename TA_, Strategy SG_, Prong NP_, typename T_>
HFSM2_CONSTEXPR(14)
bool
CS_<TN_, TA_, SG_, NP_, TL_<T_>>::wideEntryGuard(GuardControl& control,
												 const Prong HFSM2_IF_ASSERT(prong)) noexcept
{
	HFSM2_ASSERT(prong == PRONG_INDEX);

	return Single::deepEntryGuard(control);
}

template <typename TN_, typename TA_, Strategy SG_, Prong NP_, typename T_>
HFSM2_CONSTEXPR(14)
void
CS_<TN_, TA_, SG_, NP_, TL_<T_>>::wideEnter(PlanControl& control,
											const Prong HFSM2_IF_ASSERT(prong)) noexcept
{
	HFSM2_ASSERT(prong == PRONG_INDEX);

	Single::deepEnter(control);
}

template <typename TN_, typename TA_, Strategy SG_, Prong NP_, typename T_>
HFSM2_CONSTEXPR(14)
void
CS_<TN_, TA_, SG_, NP_, TL_<T_>>::wideReenter(PlanControl& control,
											  const Prong HFSM2_IF_ASSERT(prong)) noexcept
{
	HFSM2_ASSERT(prong == PRONG_INDEX);

	Single::deepReenter(control);
}

template <typename TN_, typename TA_, Strategy SG_, Prong NP_, typename T_>
HFSM2_CONSTEXPR(14)
TaskStatus
CS_<TN_, TA_, SG_, NP_, TL_<T_>>::widePreUpdate(FullControl& control,
												const Prong HFSM2_IF_ASSERT(prong)) noexcept
{
	HFSM2_ASSERT(prong == PRONG_INDEX);

	return Single::deepPreUpdate(control);
}

template <typename TN_, typename TA_, Strategy SG_, Prong NP_, typename T_>
HFSM2_CONSTEXPR(14)
TaskStatus
CS_<TN_, TA_, SG_, NP_, TL_<T_>>::wideUpdate(FullControl& control,
											 const Prong HFSM2_IF_ASSERT(prong)) noexcept
{
	HFSM2_ASSERT(prong == PRONG_INDEX);

	return Single::deepUpdate(control);
}

template <typename TN_, typename TA_, Strategy SG_, Prong NP_, typename T_>
HFSM2_CONSTEXPR(14)
TaskStatus
CS_<TN_, TA_, SG_, NP_, TL_<T_>>::widePostUpdate(FullControl& control,
												 const Prong HFSM2_IF_ASSERT(prong)) noexcept
{
	HFSM2_ASSERT(prong == PRONG_INDEX);

	return Single::deepPostUpdate(control);
}

template <typename TN_, typename TA_, Strategy SG_, Prong NP_, typename T_>
template <typename TEvent>
HFSM2_CONSTEXPR(14)
TaskStatus
CS_<TN_, TA_, SG_, NP_, TL_<T_>>::widePreReact(EventControl& control,
											   const TEvent& event,
											   const Prong HFSM2_IF_ASSERT(prong)) noexcept
{
	HFSM2_ASSERT(prong == PRONG_INDEX);

	return Single::deepPreReact(control, event);
}

template <typename TN_, typename TA_, Strategy SG_, Prong NP_, typename T_>
template <typename TEvent>
HFSM2_CONSTEXPR(14)
TaskStatus
CS_<TN_, TA_, SG_, NP_, TL_<T_>>::wideReact(EventControl& control,
											const TEvent& event,
											const Prong HFSM2_IF_ASSERT(prong)) noexcept
{
	HFSM2_ASSERT(prong == PRONG_INDEX);

	return Single::deepReact(control, event);
}

template <typename TN_, typename TA_, Strategy SG_, Prong NP_, typename T_>
template <typename TEvent>
HFSM2_CONSTEXPR(14)
TaskStatus
CS_<TN_, TA_, SG_, NP_, TL_<T_>>::widePostReact(EventControl& control,
												const TEvent& event,
												const Prong HFSM2_IF_ASSERT(prong)) noexcept
{
	HFSM2_ASSERT(prong == PRONG_INDEX);

	return Single::deepPostReact(control, event);
}

template <typename TN_, typename TA_, Strategy SG_, Prong NP_, typename T_>
template <typename TEvent>
HFSM2_CONSTEXPR(14)
void
CS_<TN_, TA_, SG_, NP_, TL_<T_>>::wideQuery(ConstControl& control,
											TEvent& event,
											const Prong HFSM2_IF_ASSERT(prong)) const noexcept
{
	HFSM2_ASSERT(prong == PRONG_INDEX);

	return Single::deepQuery(control, event);
}

#if HFSM2_PLANS_AVAILABLE()

template <typename TN_, typename TA_, Strategy SG_, Prong NP_, typename T_>
HFSM2_CONSTEXPR(14)
TaskStatus
CS_<TN_, TA_, SG_, NP_, TL_<T_>>::wideUpdatePlans(FullControl& control,
												  const Prong HFSM2_IF_ASSERT(prong)) noexcept
{
	HFSM2_ASSERT(prong == PRONG_INDEX);

	return Single::deepUpdatePlans(control);
}

#endif

template <typename TN_, typename TA_, Strategy SG_, Prong NP_, typename T_>
HFSM2_CONSTEXPR(14)
bool
CS_<TN_, TA_, SG_, NP_, TL_<T_>>::wideForwardExitGuard(GuardControl& control,
													   const Prong HFSM2_IF_ASSERT(prong)) noexcept
{
	HFSM2_ASSERT(prong == PRONG_INDEX);

	return Single::deepForwardExitGuard(control);
}

template <typename TN_, typename TA_, Strategy SG_, Prong NP_, typename T_>
HFSM2_CONSTEXPR(14)
bool
CS_<TN_, TA_, SG_, NP_, TL_<T_>>::wideExitGuard(GuardControl& control,
												const Prong HFSM2_IF_ASSERT(prong)) noexcept
{
	HFSM2_ASSERT(prong == PRONG_INDEX);

	return Single::deepExitGuard(control);
}

template <typename TN_, typename TA_, Strategy SG_, Prong NP_, typename T_>
HFSM2_CONSTEXPR(14)
void
CS_<TN_, TA_, SG_, NP_, TL_<T_>>::wideExit(PlanControl& control,
										   const Prong HFSM2_IF_ASSERT(prong)) noexcept
{
	HFSM2_ASSERT(prong == PRONG_INDEX);

	Single::deepExit(control);
}

template <typename TN_, typename TA_, Strategy SG_, Prong NP_, typename T_>
HFSM2_CONSTEXPR(14)
void
CS_<TN_, TA_, SG_, NP_, TL_<T_>>::wideForwardActive(Control& control,
													const Request request,
													const Prong HFSM2_IF_ASSERT(prong)) noexcept
{
	HFSM2_ASSERT(prong == PRONG_INDEX);

	Single::deepForwardActive(control, request);
}

template <typename TN_, typename TA_, Strategy SG_, Prong NP_, typename T_>
HFSM2_CONSTEXPR(14)
void
CS_<TN_, TA_, SG_, NP_, TL_<T_>>::wideForwardRequest(Control& control,
													 const Request request,
													 const Prong HFSM2_IF_ASSERT(prong)) noexcept
{
	HFSM2_ASSERT(prong == PRONG_INDEX);

	Single::deepForwardRequest(control, request);
}

template <typename TN_, typename TA_, Strategy SG_, Prong NP_, typename T_>
HFSM2_CONSTEXPR(14)
void
CS_<TN_, TA_, SG_, NP_, TL_<T_>>::wideRequestChangeComposite(Control& control,
															 const Request request) noexcept
{
	Single::deepRequestChange(control, request);
}

template <typename TN_, typename TA_, Strategy SG_, Prong NP_, typename T_>
HFSM2_CONSTEXPR(14)
void
CS_<TN_, TA_, SG_, NP_, TL_<T_>>::wideRequestChangeResumable(Control& control,
															 const Request request,
															 const Prong HFSM2_IF_ASSERT(prong)) noexcept
{
	HFSM2_ASSERT(prong == PRONG_INDEX);

	Single::deepRequestChange(control, request);
}

template <typename TN_, typename TA_, Strategy SG_, Prong NP_, typename T_>
HFSM2_CONSTEXPR(14)
void
CS_<TN_, TA_, SG_, NP_, TL_<T_>>::wideRequestChangeSelectable(Control& control,
															  const Request request,
															  const Prong HFSM2_IF_ASSERT(prong)) noexcept
{
	HFSM2_ASSERT(prong == PRONG_INDEX);

	Single::deepRequestChange(control, request);
}

template <typename TN_, typename TA_, Strategy SG_, Prong NP_, typename T_>
HFSM2_CONSTEXPR(14)
void
CS_<TN_, TA_, SG_, NP_, TL_<T_>>::wideRequestRestart(Control& control,
													 const Request request) noexcept
{
	Single::deepRequestRestart(control, request);
}

template <typename TN_, typename TA_, Strategy SG_, Prong NP_, typename T_>
HFSM2_CONSTEXPR(14)
void
CS_<TN_, TA_, SG_, NP_, TL_<T_>>::wideRequestResume(Control& control,
													const Request request,
													const Prong HFSM2_IF_ASSERT(prong)) noexcept
{
	HFSM2_ASSERT(prong == PRONG_INDEX);

	Single::deepRequestResume(control, request);
}

template <typename TN_, typename TA_, Strategy SG_, Prong NP_, typename T_>
HFSM2_CONSTEXPR(14)
void
CS_<TN_, TA_, SG_, NP_, TL_<T_>>::wideRequestSelect(Control& control,
													const Request request,
													const Prong HFSM2_IF_ASSERT(prong)) noexcept
{
	HFSM2_ASSERT(prong == PRONG_INDEX);

	Single::deepRequestSelect(control, request);
}

#if HFSM2_UTILITY_THEORY_AVAILABLE()

template <typename TN_, typename TA_, Strategy SG_, Prong NP_, typename T_>
HFSM2_CONSTEXPR(14)
typename TA_::UP
CS_<TN_, TA_, SG_, NP_, TL_<T_>>::wideReportUtilize(Control& control) noexcept {
	return Single::deepReportUtilize(control);
}

template <typename TN_, typename TA_, Strategy SG_, Prong NP_, typename T_>
HFSM2_CONSTEXPR(14)
typename TA_::Rank
CS_<TN_, TA_, SG_, NP_, TL_<T_>>::wideReportRank(Control& control,
												 Rank* const ranks) noexcept
{
	HFSM2_ASSERT(ranks);

*ranks = Single::deepReportRank(control);

return *ranks;
}

template <typename TN_, typename TA_, Strategy SG_, Prong NP_, typename T_>
HFSM2_CONSTEXPR(14)
typename TA_::Utility
CS_<TN_, TA_, SG_, NP_, TL_<T_>>::wideReportRandomize(Control& control,
													  Utility* const utilities,
													  const Rank* const ranks,
													  const Rank top) noexcept
{
	HFSM2_ASSERT(utilities && ranks);

*utilities = (*ranks == top) ?
	Single::deepReportRandomize(control) : Utility{0};

return *utilities;
}

template <typename TN_, typename TA_, Strategy SG_, Prong NP_, typename T_>
HFSM2_CONSTEXPR(14)
typename TA_::UP
CS_<TN_, TA_, SG_, NP_, TL_<T_>>::wideReportChangeComposite(Control& control) noexcept {
	return Single::deepReportChange(control);
}

template <typename TN_, typename TA_, Strategy SG_, Prong NP_, typename T_>
HFSM2_CONSTEXPR(14)
typename TA_::UP
CS_<TN_, TA_, SG_, NP_, TL_<T_>>::wideReportChangeResumable(Control& control,
															const Prong HFSM2_IF_ASSERT(prong)) noexcept
{
	HFSM2_ASSERT(prong == PRONG_INDEX);

	return Single::deepReportChange(control);
}

template <typename TN_, typename TA_, Strategy SG_, Prong NP_, typename T_>
HFSM2_CONSTEXPR(14)
typename TA_::UP
CS_<TN_, TA_, SG_, NP_, TL_<T_>>::wideReportChangeSelectable(Control& control,
															 const Prong HFSM2_IF_ASSERT(prong)) noexcept
{
	HFSM2_ASSERT(prong == PRONG_INDEX);

	return Single::deepReportChange(control);
}

template <typename TN_, typename TA_, Strategy SG_, Prong NP_, typename T_>
HFSM2_CONSTEXPR(14)
typename TA_::UP
CS_<TN_, TA_, SG_, NP_, TL_<T_>>::wideReportChangeUtilitarian(Control& control) noexcept {
	return Single::deepReportChange(control);
}

template <typename TN_, typename TA_, Strategy SG_, Prong NP_, typename T_>
HFSM2_CONSTEXPR(14)
typename TA_::Utility
CS_<TN_, TA_, SG_, NP_, TL_<T_>>::wideReportChangeRandom(Control& control,
														 Utility* const utilities,
														 const Rank* const ranks,
														 const Rank top) noexcept
{
	HFSM2_ASSERT(utilities && ranks);

*utilities = (*ranks == top) ?
	Single::deepReportChange(control).utility : Utility{0};

return *utilities;
}

#endif

template <typename TN_, typename TA_, Strategy SG_, Prong NP_, typename T_>
HFSM2_CONSTEXPR(14)
void
CS_<TN_, TA_, SG_, NP_, TL_<T_>>::wideChangeToRequested(PlanControl& control,
														const Prong HFSM2_IF_ASSERT(prong)) noexcept
{
	HFSM2_ASSERT(prong == PRONG_INDEX);

	Single::deepChangeToRequested(control);
}

#if HFSM2_SERIALIZATION_AVAILABLE()

template <typename TN_, typename TA_, Strategy SG_, Prong NP_, typename T_>
HFSM2_CONSTEXPR(14)
void
CS_<TN_, TA_, SG_, NP_, TL_<T_>>::wideSaveActive(const Registry& registry,
												 WriteStream& stream,
												 const Prong HFSM2_IF_ASSERT(prong)) const noexcept
{
	HFSM2_ASSERT(prong == PRONG_INDEX);

	Single::deepSaveActive(registry, stream);
}

template <typename TN_, typename TA_, Strategy SG_, Prong NP_, typename T_>
HFSM2_CONSTEXPR(14)
void
CS_<TN_, TA_, SG_, NP_, TL_<T_>>::wideSaveResumable(const Registry& registry,
													WriteStream& stream) const noexcept
{
	Single::deepSaveResumable(registry, stream);
}

template <typename TN_, typename TA_, Strategy SG_, Prong NP_, typename T_>
HFSM2_CONSTEXPR(14)
void
CS_<TN_, TA_, SG_, NP_, TL_<T_>>::wideLoadRequested(Registry& registry,
													ReadStream& stream,
													const Prong HFSM2_IF_ASSERT(prong)) const noexcept
{
	HFSM2_ASSERT(prong == PRONG_INDEX);

	Single::deepLoadRequested(registry, stream);
}

template <typename TN_, typename TA_, Strategy SG_, Prong NP_, typename T_>
HFSM2_CONSTEXPR(14)
void
	CS_<TN_, TA_, SG_, NP_, TL_<T_>>::wideLoadResumable(Registry& registry,
	ReadStream& stream) const noexcept
{
	Single::deepLoadResumable(registry, stream);
}

#endif

#if HFSM2_STRUCTURE_REPORT_AVAILABLE()

template <typename TN_, typename TA_, Strategy SG_, Prong NP_, typename T_>
HFSM2_CONSTEXPR(14)
void
CS_<TN_, TA_, SG_, NP_, TL_<T_>>::wideGetNames(const Long parent,
											   const RegionType /*region*/,
											   const Short depth,
											   StructureStateInfos& stateInfos) const noexcept
{
	Single::deepGetNames(parent, RegionType::COMPOSITE, depth, stateInfos);
}

#endif

}
}

namespace hfsm2 {
	namespace detail {

		template <
		typename TIndices
		, typename TArgs
		, Strategy TStrategy
		, typename THead
		, typename... TSubStates
		>
		struct HFSM2_EMPTY_BASES C_
		: S_<TIndices, TArgs, THead>
		, CS_<
		I_<
		TIndices::STATE_ID + 1
		, TIndices::COMPO_INDEX + 1
		, TIndices::ORTHO_INDEX
		, TIndices::ORTHO_UNIT
		>
		, TArgs
		, TStrategy
		, 0
		, TL_<TSubStates...>
		>
		{
		using Indices			= TIndices;
		static constexpr StateID  HEAD_ID	  = Indices::STATE_ID;
		static constexpr Short	  COMPO_INDEX = Indices::COMPO_INDEX;
		static constexpr Short	  ORTHO_INDEX = Indices::ORTHO_INDEX;
		static constexpr Short	  ORTHO_UNIT  = Indices::ORTHO_UNIT;

		static constexpr Strategy STRATEGY	  = TStrategy;

		static constexpr RegionID REGION_ID	  = COMPO_INDEX + ORTHO_INDEX;
		static constexpr ForkID	  COMPO_ID	  = COMPO_INDEX + 1;

		using Args				= TArgs;

#if HFSM2_UTILITY_THEORY_AVAILABLE()
		using Rank				= typename Args::Rank;
		using Utility			= typename Args::Utility;
		using UP				= typename Args::UP;
#endif

		using StateList			= typename Args::StateList;
		using RegionList		= typename Args::RegionList;

		using ReactOrder		= typename Args::ReactOrder;

		using Registry			= RegistryT<Args>;
		using StateParents		= typename Registry::StateParents;

		using ConstControl		= ConstControlT<Args>;
		using ScopedCRegion		= typename ConstControl::Region;

		using Control			= ControlT	   <Args>;
		using ScopedOrigin		= typename Control::Origin;

		using PlanControl		= PlanControlT <Args>;
		using FullControl		= FullControlT <Args>;
		using ControlLock		= typename FullControl::Lock;
		using ScopedRegion		= typename PlanControl::Region;

		using GuardControl		= GuardControlT<Args>;
		using EventControl		= EventControlT<Args>;

#if HFSM2_PLANS_AVAILABLE()
		using Plan				= typename PlanControl::Plan;
#endif

		using Head				= THead;
		using HeadState			= S_<Indices, Args, Head>;

		using SubStates			= CS_<
			I_<
			HEAD_ID + 1,
			COMPO_INDEX + 1,
			ORTHO_INDEX,
			ORTHO_UNIT
			>,
		Args,
		STRATEGY,
		0,
		TL_<TSubStates...>
		>;

		using PreReactWrapper	= PreReactWrapperT <C_, ReactOrder>;
		using ReactWrapper		= ReactWrapperT	   <C_, ReactOrder>;
		using PostReactWrapper	= PostReactWrapperT<C_, ReactOrder>;
		using QueryWrapper		= QueryWrapperT	   <C_, ReactOrder>;

		using Info				= CI_<STRATEGY, Head, TSubStates...>;
		static constexpr Short WIDTH		  = Info::WIDTH;

#if HFSM2_UTILITY_THEORY_AVAILABLE()
		using Ranks				=	 Rank[WIDTH];
		using Utilities			= Utility[WIDTH];
#endif

#if HFSM2_SERIALIZATION_AVAILABLE()
		static constexpr Short WIDTH_BITS	  = Info::WIDTH_BITS;
#endif

		static constexpr Long  REGION_SIZE	  = Info::STATE_COUNT;

#if HFSM2_SERIALIZATION_AVAILABLE()
	HFSM2_CONSTEXPR(11)	static Prong		compoRequested		  (const Registry& registry)	noexcept	{ return registry.compoRequested[COMPO_INDEX];	}
HFSM2_CONSTEXPR(11)	static Prong&		compoRequested		  (		 Registry& registry)	noexcept	{ return registry.compoRequested[COMPO_INDEX];	}

	HFSM2_CONSTEXPR(11)	static Prong		compoActive			  (const Registry& registry)	noexcept	{ return registry.compoActive	[COMPO_INDEX];	}
	HFSM2_CONSTEXPR(11)	static Prong&		compoActive			  (		 Registry& registry)	noexcept	{ return registry.compoActive	[COMPO_INDEX];	}

	HFSM2_CONSTEXPR(11)	static Prong		compoResumable		  (const Registry& registry)	noexcept	{ return registry.compoResumable[COMPO_INDEX];	}
	HFSM2_CONSTEXPR(11)	static Prong&		compoResumable		  (		 Registry& registry)	noexcept	{ return registry.compoResumable[COMPO_INDEX];	}
#endif

	HFSM2_CONSTEXPR(11)	static Prong&		compoRequested		  (		  Control& control )	noexcept	{ return control._core.registry.compoRequested[COMPO_INDEX];	}
	HFSM2_CONSTEXPR(11)	static Prong&		compoActive			  (		  Control& control )	noexcept	{ return control._core.registry.compoActive	  [COMPO_INDEX];	}
	HFSM2_CONSTEXPR(11)	static Prong		compoActive			  (	 ConstControl& control )	noexcept	{ return control._core.registry.compoActive	  [COMPO_INDEX];	}
	HFSM2_CONSTEXPR(11)	static Prong&		compoResumable		  (		  Control& control )	noexcept	{ return control._core.registry.compoResumable[COMPO_INDEX];	}

#if HFSM2_PLANS_AVAILABLE()
	HFSM2_CONSTEXPR(11)	static TaskStatus&	headStatus			  (		  Control& control )	noexcept	{ return control._core.planData.headStatuses  [REGION_ID];		}
	HFSM2_CONSTEXPR(11)	static TaskStatus&	 subStatus			  (		  Control& control )	noexcept	{ return control._core.planData.subStatuses   [REGION_ID];		}
#endif

	HFSM2_CONSTEXPR(11)	static bool			compoRemain			  (		  Control& control )	noexcept	{ return control._core.registry.compoRemains.template get<COMPO_INDEX>(); }

	HFSM2_CONSTEXPR(14)	void		deepRegister				  (	   Registry& registry, const Parent parent)			noexcept;

	HFSM2_CONSTEXPR(14)	bool		deepForwardEntryGuard		  (GuardControl& control					 )			noexcept;
	HFSM2_CONSTEXPR(14)	bool		deepEntryGuard				  (GuardControl& control					 )			noexcept;

	HFSM2_CONSTEXPR(14)	void		deepEnter					  ( PlanControl& control					 )			noexcept;
	HFSM2_CONSTEXPR(14)	void		deepReenter					  ( PlanControl& control					 )			noexcept;

	HFSM2_CONSTEXPR(14)	TaskStatus	deepPreUpdate				  ( FullControl& control					 )			noexcept;
	HFSM2_CONSTEXPR(14)	TaskStatus	deepUpdate					  ( FullControl& control					 )			noexcept;
	HFSM2_CONSTEXPR(14)	TaskStatus	deepPostUpdate				  ( FullControl& control					 )			noexcept;

	template <typename TEvent>
	HFSM2_CONSTEXPR(14)	TaskStatus	deepPreReact				  (EventControl& control, const TEvent& event)			noexcept;

	template <typename TEvent>
	HFSM2_CONSTEXPR(14)	TaskStatus	deepReact					  (EventControl& control, const TEvent& event)			noexcept;

	template <typename TEvent>
	HFSM2_CONSTEXPR(14)	TaskStatus	deepPostReact				  (EventControl& control, const TEvent& event)			noexcept;

	template <typename TEvent>
	HFSM2_CONSTEXPR(14)	void		deepQuery					  (ConstControl& control,		TEvent& event)	  const noexcept;

#if HFSM2_PLANS_AVAILABLE()
	HFSM2_CONSTEXPR(14)	TaskStatus	deepUpdatePlans				  ( FullControl& control					 )			noexcept;
#endif

	HFSM2_CONSTEXPR(14)	bool		deepForwardExitGuard		  (GuardControl& control					 )			noexcept;
	HFSM2_CONSTEXPR(14)	bool		deepExitGuard				  (GuardControl& control					 )			noexcept;

	HFSM2_CONSTEXPR(14)	void		deepExit					  ( PlanControl& control					 )			noexcept;

	HFSM2_CONSTEXPR(14)	void		deepForwardActive			  (		Control& control, const Request request)		noexcept;
	HFSM2_CONSTEXPR(14)	void		deepForwardRequest			  (		Control& control, const Request request)		noexcept;

	HFSM2_CONSTEXPR(14)	void		deepRequest					  (		Control& control, const Request request)		noexcept;

#if HFSM2_EXPLICIT_MEMBER_SPECIALIZATION_AVAILABLE()

	template <Strategy = STRATEGY>
	HFSM2_CONSTEXPR(14)	void		deepRequestChange			  (		Control& control, const Request request, const Prong = INVALID_SHORT)	noexcept;

	template <>
	HFSM2_CONSTEXPR(14)	void		deepRequestChange<Composite>  (		Control& control, const Request request, const Prong)	noexcept	{ deepRequestChangeComposite  (control, request); }

	template <>
	HFSM2_CONSTEXPR(14)	void		deepRequestChange<Resumable>  (		Control& control, const Request request, const Prong)	noexcept	{ deepRequestChangeResumable  (control, request); }

	template <>
	HFSM2_CONSTEXPR(14)	void		deepRequestChange<Selectable> (		Control& control, const Request request, const Prong)	noexcept	{ deepRequestChangeSelectable (control, request); }

#if HFSM2_UTILITY_THEORY_AVAILABLE()
	template <>
	HFSM2_CONSTEXPR(14)	void		deepRequestChange<Utilitarian>(		Control& control, const Request request, const Prong)	noexcept	{ deepRequestChangeUtilitarian(control, request); }

	template <>
	HFSM2_CONSTEXPR(14)	void		deepRequestChange<RandomUtil> (		Control& control, const Request request, const Prong)	noexcept	{ deepRequestChangeRandom	  (control, request); }
#endif

#else

	HFSM2_CONSTEXPR(14)	void		deepRequestChange			  (		Control& control, const Request request)	noexcept;

#endif

	HFSM2_CONSTEXPR(14)	void		deepRequestChangeComposite	  (		Control& control, const Request request)	noexcept;
	HFSM2_CONSTEXPR(14)	void		deepRequestChangeResumable	  (		Control& control, const Request request)	noexcept;
	HFSM2_CONSTEXPR(14)	void		deepRequestChangeSelectable	  (		Control& control, const Request request)	noexcept;

#if HFSM2_UTILITY_THEORY_AVAILABLE()
	HFSM2_CONSTEXPR(14)	void		deepRequestChangeUtilitarian  (		Control& control, const Request request)	noexcept;
	HFSM2_CONSTEXPR(14)	void		deepRequestChangeRandom		  (		Control& control, const Request request)	noexcept;
#endif

	HFSM2_CONSTEXPR(14)	void		deepRequestRestart			  (		Control& control, const Request request)	noexcept;
	HFSM2_CONSTEXPR(14)	void		deepRequestResume			  (		Control& control, const Request request)	noexcept;
	HFSM2_CONSTEXPR(14)	void		deepRequestSelect			  (		Control& control, const Request request)	noexcept;

#if HFSM2_UTILITY_THEORY_AVAILABLE()
	HFSM2_CONSTEXPR(14)	void		deepRequestUtilize			  (		Control& control, const Request request)	noexcept;
	HFSM2_CONSTEXPR(14)	void		deepRequestRandomize		  (		Control& control, const Request request)	noexcept;
#endif

#if HFSM2_UTILITY_THEORY_AVAILABLE()
#if HFSM2_EXPLICIT_MEMBER_SPECIALIZATION_AVAILABLE()

	template <Strategy = STRATEGY>
	HFSM2_CONSTEXPR(14)	UP			deepReportChange			  (		Control& control)	noexcept;

	template <>
	HFSM2_CONSTEXPR(14)	UP			deepReportChange<Composite>   (		Control& control)	noexcept	{ return deepReportChangeComposite  (control); }

	template <>
	HFSM2_CONSTEXPR(14)	UP			deepReportChange<Resumable>   (		Control& control)	noexcept	{ return deepReportChangeResumable  (control); }

	template <>
	HFSM2_CONSTEXPR(14)	UP			deepReportChange<Selectable>  (		Control& control)	noexcept	{ return deepReportChangeSelectable (control); }

	template <>
	HFSM2_CONSTEXPR(14)	UP			deepReportChange<Utilitarian> (		Control& control)	noexcept	{ return deepReportChangeUtilitarian(control); }

	template <>
	HFSM2_CONSTEXPR(14)	UP			deepReportChange<RandomUtil>  (		Control& control)	noexcept	{ return deepReportChangeRandom		(control); }

#else

	HFSM2_CONSTEXPR(14)	UP			deepReportChange			  (		Control& control)	noexcept;

#endif

	HFSM2_CONSTEXPR(14)	UP			deepReportChangeComposite	  (		Control& control)	noexcept;
	HFSM2_CONSTEXPR(14)	UP			deepReportChangeResumable	  (		Control& control)	noexcept;
	HFSM2_CONSTEXPR(14)	UP			deepReportChangeSelectable	  (		Control& control)	noexcept;
	HFSM2_CONSTEXPR(14)	UP			deepReportChangeUtilitarian   (		Control& control)	noexcept;
	HFSM2_CONSTEXPR(14)	UP			deepReportChangeRandom		  (		Control& control)	noexcept;

	HFSM2_CONSTEXPR(14)	UP			deepReportUtilize			  (		Control& control)	noexcept;
	HFSM2_CONSTEXPR(14)	Rank		deepReportRank				  (		Control& control)	noexcept;
	HFSM2_CONSTEXPR(14)	Utility		deepReportRandomize			  (		Control& control)	noexcept;

	HFSM2_CONSTEXPR(14)	Prong		resolveRandom				  (		Control& control,
																   const Utilities& utilities, const Utility sum,
																   const Ranks	  & ranks	 , const Rank	 top)  const noexcept;
#endif

	HFSM2_CONSTEXPR(14)	void		deepChangeToRequested		  ( PlanControl& control)	noexcept;

#if HFSM2_SERIALIZATION_AVAILABLE()
	using WriteStream	= typename Args::WriteStream;
	using ReadStream	= typename Args::ReadStream;

	HFSM2_CONSTEXPR(14)	void		deepSaveActive				  (const Registry& registry, WriteStream& stream)  const noexcept;
	HFSM2_CONSTEXPR(14)	void		deepSaveResumable			  (const Registry& registry, WriteStream& stream)  const noexcept;

	HFSM2_CONSTEXPR(14)	void		deepLoadRequested			  (		 Registry& registry,  ReadStream& stream)  const noexcept;
	HFSM2_CONSTEXPR(14)	void		deepLoadResumable			  (		 Registry& registry,  ReadStream& stream)  const noexcept;
#endif

#if HFSM2_STRUCTURE_REPORT_AVAILABLE()
	using StructureStateInfos = typename Args::StructureStateInfos;

	static constexpr Long NAME_COUNT = HeadState::NAME_COUNT + SubStates::NAME_COUNT;

	HFSM2_CONSTEXPR(14)	void deepGetNames(const Long parent,
										  const RegionType region,
										  const Short depth,
										  StructureStateInfos& stateInfos)  const noexcept;
#endif

};

}
}

namespace hfsm2 {
	namespace detail {

		template <typename TN_, typename TA_, Strategy SG_, typename TH_, typename... TS_>
		HFSM2_CONSTEXPR(14)
		void
		C_<TN_, TA_, SG_, TH_, TS_...>::deepRegister(Registry& registry,
		const Parent parent) noexcept
		{
		registry.compoParents[COMPO_INDEX] = parent;
		registry.regionHeads [REGION_ID]   = HEAD_ID;
		registry.regionSizes [REGION_ID]   = REGION_SIZE;

		HeadState::deepRegister(registry, parent);
		SubStates::wideRegister(registry, Parent{COMPO_ID});
	}

	template <typename TN_, typename TA_, Strategy SG_, typename TH_, typename... TS_>
	HFSM2_CONSTEXPR(14)
	bool
	C_<TN_, TA_, SG_, TH_, TS_...>::deepForwardEntryGuard(GuardControl& control) noexcept {
	const Prong	 requested	= compoRequested(control);

	const Prong	 active		= compoActive   (control);
	HFSM2_ASSERT(active		< WIDTH);

	ScopedRegion region{control, REGION_ID, HEAD_ID, REGION_SIZE};

	if (requested == INVALID_PRONG)
		return SubStates::wideForwardEntryGuard(control, active);
	else
		return SubStates::wideEntryGuard	   (control, requested);
}

template <typename TN_, typename TA_, Strategy SG_, typename TH_, typename... TS_>
HFSM2_CONSTEXPR(14)
bool
C_<TN_, TA_, SG_, TH_, TS_...>::deepEntryGuard(GuardControl& control) noexcept {
const Prong  requested = compoRequested(control);
	HFSM2_ASSERT(requested < WIDTH);

ScopedRegion region{control, REGION_ID, HEAD_ID, REGION_SIZE};

	return HeadState::deepEntryGuard(control) ||
		   SubStates::wideEntryGuard(control, requested);
}

template <typename TN_, typename TA_, Strategy SG_, typename TH_, typename... TS_>
HFSM2_CONSTEXPR(14)
void
C_<TN_, TA_, SG_, TH_, TS_...>::deepEnter(PlanControl& control) noexcept {
Prong& requested = compoRequested(control);
Prong& active	 = compoActive	 (control);
Prong& resumable = compoResumable(control);

	HFSM2_ASSERT(requested < WIDTH);
	HFSM2_ASSERT(active	  == INVALID_PRONG);

active	  = requested;

	if (requested == resumable)
resumable = INVALID_PRONG;

requested = INVALID_PRONG;

ScopedRegion region{control, REGION_ID, HEAD_ID, REGION_SIZE};

	HeadState::deepEnter(control);
	SubStates::wideEnter(control, active);
}

template <typename TN_, typename TA_, Strategy SG_, typename TH_, typename... TS_>
HFSM2_CONSTEXPR(14)
void
C_<TN_, TA_, SG_, TH_, TS_...>::deepReenter(PlanControl& control) noexcept {
Prong& requested = compoRequested(control);
Prong& active	 = compoActive   (control);
Prong& resumable = compoResumable(control);

	HFSM2_ASSERT(active	   < WIDTH &&
				 requested < WIDTH);

ScopedRegion region{control, REGION_ID, HEAD_ID, REGION_SIZE};

	HeadState::deepReenter(control);

	if (active == requested)
		SubStates::wideReenter(control, active);
	else {
		SubStates::wideExit	  (control, active);

active  = requested;

		if (requested == resumable) {
resumable = INVALID_PRONG;
		}

		SubStates::wideEnter  (control, active);
	}

requested = INVALID_PRONG;
}

template <typename TN_, typename TA_, Strategy SG_, typename TH_, typename... TS_>
HFSM2_CONSTEXPR(14)
TaskStatus
C_<TN_, TA_, SG_, TH_, TS_...>::deepPreUpdate(FullControl& control) noexcept {
	HFSM2_ASSERT(compoRequested(control) == INVALID_PRONG);

const Prong  active = compoActive(control);
	HFSM2_ASSERT(active < WIDTH);

ScopedRegion region{control, REGION_ID, HEAD_ID, REGION_SIZE};

const TaskStatus h =
	HeadState::deepPreUpdate(control);
	HFSM2_IF_PLANS(headStatus	(control) |= h);

	HFSM2_IF_PLANS( subStatus	(control) |=)
		SubStates::widePreUpdate(control, active);

return h;
}

template <typename TN_, typename TA_, Strategy SG_, typename TH_, typename... TS_>
HFSM2_CONSTEXPR(14)
TaskStatus
C_<TN_, TA_, SG_, TH_, TS_...>::deepUpdate(FullControl& control) noexcept {
	HFSM2_ASSERT(compoRequested(control) == INVALID_PRONG);

const Prong  active = compoActive(control);
	HFSM2_ASSERT(active < WIDTH);

ScopedRegion region{control, REGION_ID, HEAD_ID, REGION_SIZE};

const TaskStatus h =
	HeadState::deepUpdate(control);
	HFSM2_IF_PLANS(headStatus(control) |= h);

	HFSM2_IF_PLANS( subStatus(control) |=)
		SubStates::wideUpdate(control, active);

return h;
}

template <typename TN_, typename TA_, Strategy SG_, typename TH_, typename... TS_>
HFSM2_CONSTEXPR(14)
TaskStatus
C_<TN_, TA_, SG_, TH_, TS_...>::deepPostUpdate(FullControl& control) noexcept {
	HFSM2_ASSERT(compoRequested(control) == INVALID_PRONG);

const Prong  active = compoActive(control);
	HFSM2_ASSERT(active < WIDTH);

ScopedRegion region{control, REGION_ID, HEAD_ID, REGION_SIZE};

	HFSM2_IF_PLANS( subStatus	 (control) |=)
		SubStates::widePostUpdate(control, active);

const TaskStatus h =
	HeadState::deepPostUpdate(control);
	HFSM2_IF_PLANS(headStatus	 (control) |= h);

return h;
}

template <typename TN_, typename TA_, Strategy SG_, typename TH_, typename... TS_>
template <typename TEvent>
HFSM2_CONSTEXPR(14)
TaskStatus
C_<TN_, TA_, SG_, TH_, TS_...>::deepPreReact(EventControl& control,
											 const TEvent& event) noexcept
{
	HFSM2_ASSERT(compoRequested(control) == INVALID_PRONG);

const Prong  active = compoActive(control);
	HFSM2_ASSERT(active < WIDTH);

ScopedRegion region{control, REGION_ID, HEAD_ID, REGION_SIZE};

	return PreReactWrapper::execute(*this, control, event, active);
}

template <typename TN_, typename TA_, Strategy SG_, typename TH_, typename... TS_>
template <typename TEvent>
HFSM2_CONSTEXPR(14)
TaskStatus
C_<TN_, TA_, SG_, TH_, TS_...>::deepReact(EventControl& control,
										  const TEvent& event) noexcept
{
	HFSM2_ASSERT(compoRequested(control) == INVALID_PRONG);

const Prong  active = compoActive(control);
	HFSM2_ASSERT(active < WIDTH);

ScopedRegion region{control, REGION_ID, HEAD_ID, REGION_SIZE};

	return ReactWrapper::execute(*this, control, event, active);
}

template <typename TN_, typename TA_, Strategy SG_, typename TH_, typename... TS_>
template <typename TEvent>
HFSM2_CONSTEXPR(14)
TaskStatus
C_<TN_, TA_, SG_, TH_, TS_...>::deepPostReact(EventControl& control,
											  const TEvent& event) noexcept
{
	HFSM2_ASSERT(compoRequested(control) == INVALID_PRONG);

const Prong  active = compoActive(control);
	HFSM2_ASSERT(active < WIDTH);

ScopedRegion region{control, REGION_ID, HEAD_ID, REGION_SIZE};

	return PostReactWrapper::execute(*this, control, event, active);
}

template <typename TN_, typename TA_, Strategy SG_, typename TH_, typename... TS_>
template <typename TEvent>
HFSM2_CONSTEXPR(14)
void
C_<TN_, TA_, SG_, TH_, TS_...>::deepQuery(ConstControl& control,
										  TEvent& event) const noexcept
{
const Prong  active = compoActive(control);
	HFSM2_ASSERT(active < WIDTH);

ScopedCRegion region{control, REGION_ID};

	QueryWrapper::execute(*this, control, event, active);
}

#if HFSM2_PLANS_AVAILABLE()

template <typename TN_, typename TA_, Strategy SG_, typename TH_, typename... TS_>
HFSM2_CONSTEXPR(14)
TaskStatus
C_<TN_, TA_, SG_, TH_, TS_...>::deepUpdatePlans(FullControl& control) noexcept {
	HFSM2_ASSERT(compoRequested(control) == INVALID_PRONG);

const Prong  active = compoActive(control);
	HFSM2_ASSERT(active < WIDTH);

const TaskStatus h = headStatus(control) |
	HeadState::deepUpdatePlans (control);

const TaskStatus s =  subStatus(control) |
	SubStates::wideUpdatePlans (control, active);

	if (h)
return h;
	else {
		if (s.outerTransition)
return TaskStatus{TaskStatus::NONE, true};

ScopedRegion region{control, REGION_ID, HEAD_ID, REGION_SIZE};

const bool planExists = control._core.planData.planExists.template get<REGION_ID>();

		return s && planExists ?
			control.updatePlan(static_cast<HeadState&>(*this), s) : s;
	}
}

#endif

template <typename TN_, typename TA_, Strategy SG_, typename TH_, typename... TS_>
HFSM2_CONSTEXPR(14)
bool
C_<TN_, TA_, SG_, TH_, TS_...>::deepForwardExitGuard(GuardControl& control) noexcept {
const Prong  active = compoActive(control);
	HFSM2_ASSERT(active < WIDTH);

ScopedRegion region{control, REGION_ID, HEAD_ID, REGION_SIZE};

	if (compoRequested(control) == INVALID_PRONG)
		return SubStates::wideForwardExitGuard(control, active);
	else
		return SubStates::wideExitGuard		  (control, active);
}

template <typename TN_, typename TA_, Strategy SG_, typename TH_, typename... TS_>
HFSM2_CONSTEXPR(14)
bool
C_<TN_, TA_, SG_, TH_, TS_...>::deepExitGuard(GuardControl& control) noexcept {
const Prong  active = compoActive(control);
	HFSM2_ASSERT(active < WIDTH);

ScopedRegion region{control, REGION_ID, HEAD_ID, REGION_SIZE};

	return SubStates::wideExitGuard(control, active) ||
		   HeadState::deepExitGuard(control);
}

template <typename TN_, typename TA_, Strategy SG_, typename TH_, typename... TS_>
HFSM2_CONSTEXPR(14)
void
C_<TN_, TA_, SG_, TH_, TS_...>::deepExit(PlanControl& control) noexcept {
Prong& active	 = compoActive   (control);
	HFSM2_ASSERT(active < WIDTH);

Prong& resumable = compoResumable(control);

	SubStates::wideExit(control, active);
	HeadState::deepExit(control);

resumable = active;
active	  = INVALID_PRONG;
}

template <typename TN_, typename TA_, Strategy SG_, typename TH_, typename... TS_>
HFSM2_CONSTEXPR(14)
void
C_<TN_, TA_, SG_, TH_, TS_...>::deepForwardActive(Control& control,
												  const Request request) noexcept
{
	HFSM2_ASSERT(HEAD_ID == ROOT_ID || control._core.registry.isActive(HEAD_ID));

const Prong requested = compoRequested(control);

	if (requested == INVALID_SHORT) {
const Prong active = compoActive(control);

		SubStates::wideForwardActive (control, request, active);
	} else
		SubStates::wideForwardRequest(control, request, requested);
}

template <typename TN_, typename TA_, Strategy SG_, typename TH_, typename... TS_>
HFSM2_CONSTEXPR(14)
void
C_<TN_, TA_, SG_, TH_, TS_...>::deepForwardRequest(Control& control,
												   const Request request) noexcept
{
	HFSM2_IF_TRANSITION_HISTORY(control.pinLastTransition(HEAD_ID, request.index));

const Prong requested = compoRequested(control);

	if (requested != INVALID_PRONG)
		SubStates::wideForwardRequest(control, request, requested);
	else
		deepRequest					 (control, request);
}

template <typename TN_, typename TA_, Strategy SG_, typename TH_, typename... TS_>
void
HFSM2_CONSTEXPR(14)
C_<TN_, TA_, SG_, TH_, TS_...>::deepRequest(Control& control,
											const Request request) noexcept
{
	switch (request.type) {
	case TransitionType::CHANGE:
		deepRequestChange	(control, request);
		break;

	case TransitionType::RESTART:
		deepRequestRestart	(control, request);
		break;

	case TransitionType::RESUME:
		deepRequestResume	(control, request);
		break;

	case TransitionType::SELECT:
		deepRequestSelect	(control, request);
		break;

#if HFSM2_UTILITY_THEORY_AVAILABLE()

	case TransitionType::UTILIZE:
		deepRequestUtilize	(control, request);
		break;

	case TransitionType::RANDOMIZE:
		deepRequestRandomize(control, request);
		break;

#endif

	default:
		HFSM2_BREAK();
	}
}

#if !HFSM2_EXPLICIT_MEMBER_SPECIALIZATION_AVAILABLE()

template <typename TN_, typename TA_, Strategy SG_, typename TH_, typename... TS_>
HFSM2_CONSTEXPR(14)
void
C_<TN_, TA_, SG_, TH_, TS_...>::deepRequestChange(Control& control,
												  const Request request) noexcept
{
	switch (STRATEGY) {
	case Strategy::Composite:
		deepRequestChangeComposite  (control, request);
		break;

	case Strategy::Resumable:
		deepRequestChangeResumable  (control, request);
		break;

	case Strategy::Selectable:
		deepRequestChangeSelectable	(control, request);
		break;

#if HFSM2_UTILITY_THEORY_AVAILABLE()

	case Strategy::Utilitarian:
		deepRequestChangeUtilitarian(control, request);
		break;

	case Strategy::RandomUtil:
		deepRequestChangeRandom		(control, request);
		break;

#endif

	default:
		HFSM2_BREAK();
	}
}

#endif

template <typename TN_, typename TA_, Strategy SG_, typename TH_, typename... TS_>
HFSM2_CONSTEXPR(14)
void
C_<TN_, TA_, SG_, TH_, TS_...>::deepRequestChangeComposite(Control& control,
														   const Request request) noexcept
{
	HFSM2_IF_TRANSITION_HISTORY(control.pinLastTransition(HEAD_ID, request.index));

Prong& requested = compoRequested(control);

requested = 0;

	SubStates::wideRequestChangeComposite(control, request);
}

template <typename TN_, typename TA_, Strategy SG_, typename TH_, typename... TS_>
HFSM2_CONSTEXPR(14)
void
C_<TN_, TA_, SG_, TH_, TS_...>::deepRequestChangeResumable(Control& control,
														   const Request request) noexcept
{
	HFSM2_IF_TRANSITION_HISTORY(control.pinLastTransition(HEAD_ID, request.index));

Prong& requested = compoRequested(control);
const Prong  resumable = compoResumable(control);

requested = (resumable != INVALID_PRONG) ?
	resumable : 0;

	HFSM2_ASSERT(requested < WIDTH);

	SubStates::wideRequestChangeResumable(control, request, requested);
}

template <typename TN_, typename TA_, Strategy SG_, typename TH_, typename... TS_>
HFSM2_CONSTEXPR(14)
void
C_<TN_, TA_, SG_, TH_, TS_...>::deepRequestChangeSelectable(Control& control,
															const Request HFSM2_IF_TRANSITION_HISTORY(request)) noexcept
{
	HFSM2_IF_TRANSITION_HISTORY(control.pinLastTransition(HEAD_ID, request.index));

Prong& requested = compoRequested(control);
requested = HeadState::wrapSelect(control);

	HFSM2_ASSERT(requested < WIDTH);

	HFSM2_LOG_SELECT_RESOLUTION(control.context(), HEAD_ID, requested);
}

#if HFSM2_UTILITY_THEORY_AVAILABLE()

template <typename TN_, typename TA_, Strategy SG_, typename TH_, typename... TS_>
HFSM2_CONSTEXPR(14)
void
C_<TN_, TA_, SG_, TH_, TS_...>::deepRequestChangeUtilitarian(Control& control,
															 const Request HFSM2_IF_TRANSITION_HISTORY(request)) noexcept
{
	HFSM2_IF_TRANSITION_HISTORY(control.pinLastTransition(HEAD_ID, request.index));

const UP s = SubStates::wideReportChangeUtilitarian(control);
	HFSM2_ASSERT(s.prong < WIDTH);

Prong& requested = compoRequested(control);
requested = s.prong;

	HFSM2_LOG_UTILITY_RESOLUTION(control.context(), HEAD_ID, requested, s.utility);
}

template <typename TN_, typename TA_, Strategy SG_, typename TH_, typename... TS_>
HFSM2_CONSTEXPR(14)
void
C_<TN_, TA_, SG_, TH_, TS_...>::deepRequestChangeRandom(Control& control,
														const Request HFSM2_IF_TRANSITION_HISTORY(request)) noexcept
{
	HFSM2_IF_TRANSITION_HISTORY(control.pinLastTransition(HEAD_ID, request.index));

Rank ranks[WIDTH] = { Rank{} };
Rank top = SubStates::wideReportRank(control, ranks);

Utility utilities[WIDTH] = { Utility{} };
const UP sum = SubStates::wideReportChangeRandom(control, utilities, ranks, top);

Prong& requested = compoRequested(control);
requested = resolveRandom(control, utilities, sum.utility, ranks, top);
	HFSM2_ASSERT(requested < WIDTH);
}

#endif

template <typename TN_, typename TA_, Strategy SG_, typename TH_, typename... TS_>
HFSM2_CONSTEXPR(14)
void
C_<TN_, TA_, SG_, TH_, TS_...>::deepRequestRestart(Control& control,
												   const Request request) noexcept
{
	HFSM2_IF_TRANSITION_HISTORY(control.pinLastTransition(HEAD_ID, request.index));

Prong& requested = compoRequested(control);

requested = 0;

	SubStates::wideRequestRestart(control, request);
}

template <typename TN_, typename TA_, Strategy SG_, typename TH_, typename... TS_>
HFSM2_CONSTEXPR(14)
void
C_<TN_, TA_, SG_, TH_, TS_...>::deepRequestResume(Control& control,
												  const Request request) noexcept
{
	HFSM2_IF_TRANSITION_HISTORY(control.pinLastTransition(HEAD_ID, request.index));

Prong& requested = compoRequested(control);
const Prong  resumable = compoResumable(control);

requested = (resumable != INVALID_PRONG) ?
	resumable : 0;

	HFSM2_ASSERT(requested < WIDTH);

	SubStates::wideRequestResume(control, request, requested);
}

template <typename TN_, typename TA_, Strategy SG_, typename TH_, typename... TS_>
HFSM2_CONSTEXPR(14)
void
C_<TN_, TA_, SG_, TH_, TS_...>::deepRequestSelect(Control& control,
												  const Request HFSM2_IF_TRANSITION_HISTORY(request)) noexcept
{
	HFSM2_IF_TRANSITION_HISTORY(control.pinLastTransition(HEAD_ID, request.index));

Prong& requested = compoRequested(control);
requested = HeadState::wrapSelect(control);

	HFSM2_ASSERT(requested < WIDTH);

	HFSM2_LOG_SELECT_RESOLUTION(control.context(), HEAD_ID, requested);
}

#if HFSM2_UTILITY_THEORY_AVAILABLE()

template <typename TN_, typename TA_, Strategy SG_, typename TH_, typename... TS_>
HFSM2_CONSTEXPR(14)
void
C_<TN_, TA_, SG_, TH_, TS_...>::deepRequestUtilize(Control& control,
												   const Request HFSM2_IF_TRANSITION_HISTORY(request)) noexcept
{
	HFSM2_IF_TRANSITION_HISTORY(control.pinLastTransition(HEAD_ID, request.index));

const UP s = SubStates::wideReportUtilize(control);

Prong& requested = compoRequested(control);
requested = s.prong;

	HFSM2_ASSERT(s.prong < WIDTH);

	HFSM2_LOG_UTILITY_RESOLUTION(control.context(), HEAD_ID, requested, s.utility);
}

template <typename TN_, typename TA_, Strategy SG_, typename TH_, typename... TS_>
HFSM2_CONSTEXPR(14)
void
C_<TN_, TA_, SG_, TH_, TS_...>::deepRequestRandomize(Control& control,
													 const Request HFSM2_IF_TRANSITION_HISTORY(request)) noexcept
{
	HFSM2_IF_TRANSITION_HISTORY(control.pinLastTransition(HEAD_ID, request.index));

Rank ranks[WIDTH] = { Rank{} };
Rank top = SubStates::wideReportRank(control, ranks);

Utility utilities[WIDTH] = { Utility{} };
const Utility sum = SubStates::wideReportRandomize(control, utilities, ranks, top);

Prong& requested = compoRequested(control);
requested = resolveRandom(control, utilities, sum, ranks, top);
	HFSM2_ASSERT(requested < WIDTH);
}

#endif

#if HFSM2_UTILITY_THEORY_AVAILABLE()
#if !HFSM2_EXPLICIT_MEMBER_SPECIALIZATION_AVAILABLE()

template <typename TN_, typename TA_, Strategy SG_, typename TH_, typename... TS_>
HFSM2_CONSTEXPR(14)
typename TA_::UP
C_<TN_, TA_, SG_, TH_, TS_...>::deepReportChange(Control& control) noexcept {
	switch (STRATEGY) {
	case Strategy::Composite:
		return deepReportChangeComposite  (control);

	case Strategy::Resumable:
		return deepReportChangeResumable  (control);

	case Strategy::Selectable:
		return deepReportChangeSelectable (control);

	case Strategy::Utilitarian:
		return deepReportChangeUtilitarian(control);

	case Strategy::RandomUtil:
		return deepReportChangeRandom	  (control);

	default:
		HFSM2_BREAK();
		return UP{};
	}
}

#endif

template <typename TN_, typename TA_, Strategy SG_, typename TH_, typename... TS_>
HFSM2_CONSTEXPR(14)
typename TA_::UP
C_<TN_, TA_, SG_, TH_, TS_...>::deepReportChangeComposite(Control& control) noexcept {
Prong& requested = compoRequested(control);
requested = 0;

const UP h = HeadState::deepReportChange(control);
const UP s = SubStates::wideReportChangeComposite(control);

	return {
h.utility * s.utility,
		h.prong
	};
}

template <typename TN_, typename TA_, Strategy SG_, typename TH_, typename... TS_>
HFSM2_CONSTEXPR(14)
Short
C_<TN_, TA_, SG_, TH_, TS_...>::resolveRandom(Control& control,
											  const Utilities& utilities,
											  const Utility sum,
											  const Ranks& ranks,
											  const Rank top) const noexcept
{
const Utility random = control._core.rng.next();
	HFSM2_ASSERT(0.0f <= random && random < 1.0f);

Utility cursor = random * sum;

for (Prong i = 0; i < count<Prong>(ranks); ++i)
if (ranks[i] == top) {
			HFSM2_ASSERT(utilities[i] >= 0.0f);

if (cursor >= utilities[i])
cursor -= utilities[i];
			else {
				HFSM2_LOG_RANDOM_RESOLUTION(control.context(), HEAD_ID, i, random);

return i;
			}
		}

	HFSM2_BREAK();
return INVALID_PRONG;
}

template <typename TN_, typename TA_, Strategy SG_, typename TH_, typename... TS_>
HFSM2_CONSTEXPR(14)
typename TA_::UP
C_<TN_, TA_, SG_, TH_, TS_...>::deepReportChangeResumable(Control& control) noexcept {
const Prong  resumable = compoResumable(control);
Prong& requested = compoRequested(control);

requested = (resumable != INVALID_PRONG) ?
	resumable : 0;

const UP h = HeadState::deepReportChange(control);
const UP s = SubStates::wideReportChangeResumable(control, requested);

	return {
h.utility * s.utility,
		h.prong
	};
}

template <typename TN_, typename TA_, Strategy SG_, typename TH_, typename... TS_>
HFSM2_CONSTEXPR(14)
typename TA_::UP
C_<TN_, TA_, SG_, TH_, TS_...>::deepReportChangeSelectable(Control& control) noexcept {
const Prong  resumable = compoResumable(control);
Prong& requested = compoRequested(control);

requested = (resumable != INVALID_PRONG) ?
	resumable : 0;

	HFSM2_ASSERT(requested < WIDTH);

const UP h = HeadState::deepReportChange		  (control);
const UP s = SubStates::wideReportChangeSelectable(control, requested);

	return {
h.utility * s.utility,
		h.prong
	};
}

template <typename TN_, typename TA_, Strategy SG_, typename TH_, typename... TS_>
HFSM2_CONSTEXPR(14)
typename TA_::UP
C_<TN_, TA_, SG_, TH_, TS_...>::deepReportChangeUtilitarian(Control& control) noexcept {
const UP h = HeadState::deepReportChange(control);
const UP s = SubStates::wideReportChangeUtilitarian(control);

Prong& requested = compoRequested(control);
requested = s.prong;

	HFSM2_LOG_UTILITY_RESOLUTION(control.context(), HEAD_ID, requested, s.utility);

	return {
h.utility * s.utility,
		h.prong
	};
}

template <typename TN_, typename TA_, Strategy SG_, typename TH_, typename... TS_>
HFSM2_CONSTEXPR(14)
typename TA_::UP
C_<TN_, TA_, SG_, TH_, TS_...>::deepReportChangeRandom(Control& control) noexcept {
const UP h = HeadState::deepReportChange(control);

Rank ranks[WIDTH] = { Rank{} };
Rank top = SubStates::wideReportRank(control, ranks);

Utility utilities[WIDTH] = { Utility{} };
const UP sum = SubStates::wideReportChangeRandom(control, utilities, ranks, top);

Prong& requested = compoRequested(control);
requested = resolveRandom(control, utilities, sum.utility, ranks, top);
	HFSM2_ASSERT(requested < WIDTH);

	return {
h.utility * utilities[requested],
		h.prong
	};
}

template <typename TN_, typename TA_, Strategy SG_, typename TH_, typename... TS_>
HFSM2_CONSTEXPR(14)
typename TA_::UP
C_<TN_, TA_, SG_, TH_, TS_...>::deepReportUtilize(Control& control) noexcept {
const UP h = HeadState::deepReportUtilize(control);
const UP s = SubStates::wideReportUtilize(control);

Prong& requested = compoRequested(control);
requested = s.prong;

	HFSM2_LOG_UTILITY_RESOLUTION(control.context(), HEAD_ID, requested, s.utility);

	return {
h.utility * s.utility,
		h.prong
	};
}

template <typename TN_, typename TA_, Strategy SG_, typename TH_, typename... TS_>
HFSM2_CONSTEXPR(14)
typename TA_::Rank
C_<TN_, TA_, SG_, TH_, TS_...>::deepReportRank(Control& control) noexcept {
	return HeadState::wrapRank(control);
}

template <typename TN_, typename TA_, Strategy SG_, typename TH_, typename... TS_>
HFSM2_CONSTEXPR(14)
typename TA_::Utility
C_<TN_, TA_, SG_, TH_, TS_...>::deepReportRandomize(Control& control) noexcept {
const Utility h = HeadState::wrapUtility(control);

Rank ranks[WIDTH] = { Rank{} };
Rank top = SubStates::wideReportRank(control, ranks);

Utility utilities[WIDTH] = { Utility{} };
const Utility sum = SubStates::wideReportRandomize(control, utilities, ranks, top);

Prong& requested = compoRequested(control);
requested = resolveRandom(control, utilities, sum, ranks, top);
	HFSM2_ASSERT(requested < WIDTH);

return h * utilities[requested];
}

#endif

template <typename TN_, typename TA_, Strategy SG_, typename TH_, typename... TS_>
HFSM2_CONSTEXPR(14)
void
C_<TN_, TA_, SG_, TH_, TS_...>::deepChangeToRequested(PlanControl& control) noexcept {
Prong& requested = compoRequested(control);
Prong& active	 = compoActive	 (control);
Prong& resumable = compoResumable(control);

	HFSM2_ASSERT(active < WIDTH);

ScopedRegion region{control, REGION_ID, HEAD_ID, REGION_SIZE};

	if (requested == INVALID_PRONG)
		SubStates::wideChangeToRequested(control, active);
	else if (requested != active) {
		SubStates::wideExit	  (control, active);

		HFSM2_ASSERT(requested < WIDTH);

resumable = active;
active	  = requested;
requested = INVALID_PRONG;

		SubStates::wideEnter  (control, active);
	} else if (compoRemain(control)) {
		SubStates::wideExit   (control, active);

requested = INVALID_PRONG;

		SubStates::wideEnter  (control, active);
	} else {
requested = INVALID_PRONG;

		// reconstruction done in S_::reenter()
		SubStates::wideReenter(control, active);
	}
}

#if HFSM2_SERIALIZATION_AVAILABLE()

template <typename TN_, typename TA_, Strategy SG_, typename TH_, typename... TS_>
HFSM2_CONSTEXPR(14)
void
C_<TN_, TA_, SG_, TH_, TS_...>::deepSaveActive(const Registry& registry,
											   WriteStream& stream) const noexcept
{
const Prong active	  = compoActive   (registry);
const Prong resumable = compoResumable(registry);

	stream.template write<WIDTH_BITS>(active);

	if (resumable != INVALID_PRONG) {
		stream.template write<1>(1);
		stream.template write<WIDTH_BITS>(resumable);
	} else
		stream.template write<1>(0);

	SubStates::wideSaveActive(registry,stream, active);
}

template <typename TN_, typename TA_, Strategy SG_, typename TH_, typename... TS_>
HFSM2_CONSTEXPR(14)
void
C_<TN_, TA_, SG_, TH_, TS_...>::deepSaveResumable(const Registry& registry,
												  WriteStream& stream) const noexcept
{
const Prong resumable = compoResumable(registry);

	if (resumable != INVALID_PRONG) {
		stream.template write<1>(1);
		stream.template write<WIDTH_BITS>(resumable);
	} else
		stream.template write<1>(0);

	SubStates::wideSaveResumable(registry, stream);
}

template <typename TN_, typename TA_, Strategy SG_, typename TH_, typename... TS_>
HFSM2_CONSTEXPR(14)
void
C_<TN_, TA_, SG_, TH_, TS_...>::deepLoadRequested(Registry& registry,
												  ReadStream& stream) const noexcept
{
Prong& resumable = compoResumable(registry);
Prong& requested = compoRequested(registry);

requested = stream.template read<WIDTH_BITS>();
	HFSM2_ASSERT(requested < WIDTH);

	if (stream.template read<1>()) {
resumable = stream.template read<WIDTH_BITS>();
		HFSM2_ASSERT(resumable < WIDTH);
	} else
resumable = INVALID_PRONG;

	SubStates::wideLoadRequested(registry, stream, requested);
}

template <typename TN_, typename TA_, Strategy SG_, typename TH_, typename... TS_>
HFSM2_CONSTEXPR(14)
void
C_<TN_, TA_, SG_, TH_, TS_...>::deepLoadResumable(Registry& registry,
												  ReadStream& stream) const noexcept
{
Prong& resumable = compoResumable(registry);

	if (stream.template read<1>()) {
resumable = stream.template read<WIDTH_BITS>();
		HFSM2_ASSERT(resumable < WIDTH);
	} else
resumable = INVALID_PRONG;

	SubStates::wideLoadResumable(registry, stream);
}

#endif

#if HFSM2_STRUCTURE_REPORT_AVAILABLE()

template <typename TN_, typename TA_, Strategy SG_, typename TH_, typename... TS_>
HFSM2_CONSTEXPR(14)
void
C_<TN_, TA_, SG_, TH_, TS_...>::deepGetNames(const Long parent,
											 const RegionType regionType,
											 const Short depth,
											 StructureStateInfos& stateInfos) const noexcept
{
	HeadState::deepGetNames(parent,					regionType,			   depth,	  stateInfos);
	SubStates::wideGetNames(stateInfos.count() - 1, RegionType::COMPOSITE, depth + 1, stateInfos);
}

#endif

}
}

namespace hfsm2 {
	namespace detail {

		template <
		typename
		, typename
		, Short
		, typename...
		>
		struct OS_;

		template <
		typename TIndices
		, typename TArgs
		, Prong NProng
		, typename TInitial
		, typename... TRemaining
		>
		struct HFSM2_EMPTY_BASES OS_<
		TIndices
		, TArgs
		, NProng
		, TInitial
		, TRemaining...
		>
		:					 InitialOS<
		TIndices
		, TArgs
		, TInitial
		>
		,					 RemainingOS<
		TIndices
		, TArgs
		, NProng
		, TInitial
		, TRemaining...
		>
		{
		using Indices		= TIndices;
		static constexpr StateID INITIAL_ID	 = Indices::STATE_ID;
		static constexpr Short	 COMPO_INDEX = Indices::COMPO_INDEX;
		static constexpr Short	 ORTHO_INDEX = Indices::ORTHO_INDEX;
		static constexpr Short	 ORTHO_UNIT	 = Indices::ORTHO_UNIT;

		static constexpr Prong	 PRONG_INDEX = NProng;

		using Args			= TArgs;

#if HFSM2_UTILITY_THEORY_AVAILABLE()
		using Rank			= typename Args::Rank;
		using Utility		= typename Args::Utility;
		using UP			= typename Args::UP;
#endif

		using Registry		= RegistryT<Args>;
		using StateParents	= typename Registry::StateParents;
		using OrthoForks	= typename Registry::OrthoForks;
		using ProngBits		= typename OrthoForks::Bits;
		using ProngCBits	= typename OrthoForks::CBits;

		using ConstControl	= ConstControlT<Args>;
		using Control		= ControlT	   <Args>;
		using PlanControl	= PlanControlT <Args>;
		using FullControl	= FullControlT <Args>;
		using GuardControl	= GuardControlT<Args>;
		using EventControl	= EventControlT<Args>;

		using InitialInfo	= WrapInfo<TInitial>;
		using InitialStates	= typename InitialInfo::StateList;

		using Initial		= InitialOS<
			TIndices,
			TArgs,
			TInitial
			>;

		using Remaining		= RemainingOS<
			TIndices,
			TArgs,
			NProng,
			TInitial,
			TRemaining...
		>;

		HFSM2_CONSTEXPR(14)	void		wideRegister		 (Registry& registry, const ForkID forkId)										noexcept;

		HFSM2_CONSTEXPR(14)	bool		wideForwardEntryGuard(GuardControl& control,						const ProngCBits prongs)		noexcept;
		HFSM2_CONSTEXPR(14)	bool		wideForwardEntryGuard(GuardControl& control												   )		noexcept;
		HFSM2_CONSTEXPR(14)	bool		wideEntryGuard		 (GuardControl& control												   )		noexcept;

		HFSM2_CONSTEXPR(14)	void		wideEnter			 ( PlanControl& control												   )		noexcept;
		HFSM2_CONSTEXPR(14)	void		wideReenter			 ( PlanControl& control												   )		noexcept;

		HFSM2_CONSTEXPR(14)	TaskStatus	widePreUpdate		 ( FullControl& control												   )		noexcept;
		HFSM2_CONSTEXPR(14)	TaskStatus	wideUpdate			 ( FullControl& control												   )		noexcept;
		HFSM2_CONSTEXPR(14)	TaskStatus	widePostUpdate		 ( FullControl& control												   )		noexcept;

		template <typename TEvent>
		HFSM2_CONSTEXPR(14)	TaskStatus	widePreReact		 (EventControl& control, const TEvent& event						   )		noexcept;

		template <typename TEvent>
		HFSM2_CONSTEXPR(14)	TaskStatus	wideReact			 (EventControl& control, const TEvent& event						   )		noexcept;

		template <typename TEvent>
		HFSM2_CONSTEXPR(14)	TaskStatus	widePostReact		 (EventControl& control, const TEvent& event						   )		noexcept;

		template <typename TEvent>
		HFSM2_CONSTEXPR(14)	void		wideQuery			 (ConstControl& control,	   TEvent& event						   )  const noexcept;
```
